LIN {X 0,Y 516.884,Z 407.102,A -85,B 0,C 180,E1 -5001.284,E2 -5001.284} C_VEL
LIN {X 0,Y 516.874,Z 407.103,A -85,B 0,C 180,E1 -5004.22,E2 -5004.22} C_VEL
LIN {X 0,Y 516.899,Z 407.102,A -85,B 0,C 180,E1 -5007.053,E2 -5007.053} C_VEL
LIN {X 0,Y 516.896,Z 407.098,A -85,B 0,C 180,E1 -5009.796,E2 -5009.796} C_VEL
LIN {X 0,Y 516.931,Z 407.097,A -85,B 0,C 180,E1 -5012.467,E2 -5012.467} C_VEL
LIN {X 0,Y 516.878,Z 407.102,A -85,B 0,C 180,E1 -5015.07,E2 -5015.07} C_VEL
LIN {X 0,Y 516.871,Z 407.103,A -85,B 0,C 180,E1 -5017.621,E2 -5017.621} C_VEL
LIN {X 0,Y 516.936,Z 407.096,A -85,B 0,C 180,E1 -5020.13,E2 -5020.13} C_VEL
LIN {X 0,Y 516.935,Z 407.096,A -85,B 0,C 180,E1 -5022.596,E2 -5022.596} C_VEL
LIN {X 0,Y 516.946,Z 407.095,A -85,B 0,C 180,E1 -5025.03,E2 -5025.03} C_VEL
LIN {X 0,Y 517.008,Z 407.087,A -85,B 0,C 180,E1 -5028.235,E2 -5028.235} C_VEL
LIN {X 0,Y 516.961,Z 407.092,A -85,B 0,C 180,E1 -5031.399,E2 -5031.399} C_VEL
LIN {X 0,Y 517.013,Z 407.086,A -85,B 0,C 180,E1 -5033.757,E2 -5033.757} C_VEL
LIN {X 0,Y 517.087,Z 407.075,A -85,B 0,C 180,E1 -5037.663,E2 -5037.663} C_VEL
LIN {X 0,Y 517.098,Z 407.076,A -85,B 0,C 180,E1 -5040.779,E2 -5040.779} C_VEL
LIN {X 0,Y 517.019,Z 407.085,A -85,B 0,C 180,E1 -5043.117,E2 -5043.117} C_VEL
LIN {X 0,Y 517.014,Z 407.087,A -85,B 0,C 180,E1 -5046.243,E2 -5046.243} C_VEL
LIN {X 0,Y 516.945,Z 407.094,A -85,B 0,C 180,E1 -5049.389,E2 -5049.389} C_VEL
LIN {X 0,Y 516.987,Z 407.09,A -85,B 0,C 180,E1 -5051.824,E2 -5051.824} C_VEL
LIN {X 0,Y 516.948,Z 407.092,A -85,B 0,C 180,E1 -5055.147,E2 -5055.147} C_VEL
LIN {X 0,Y 516.93,Z 407.097,A -85,B 0,C 180,E1 -5058.222,E2 -5058.222} C_VEL
LIN {X 0,Y 516.916,Z 407.097,A -85,B 0,C 180,E1 -5060.701,E2 -5060.701} C_VEL
LIN {X 0,Y 516.893,Z 407.101,A -85,B 0,C 180,E1 -5064.073,E2 -5064.073} C_VEL
LIN {X 0,Y 516.929,Z 407.095,A -85,B 0,C 180,E1 -5066.658,E2 -5066.658} C_VEL
LIN {X 0,Y 516.914,Z 407.098,A -85,B 0,C 180,E1 -5069.524,E2 -5069.524} C_VEL
LIN {X 0,Y 516.904,Z 407.1,A -85,B 0,C 180,E1 -5072.544,E2 -5072.544} C_VEL
LIN {X 0,Y 516.884,Z 407.101,A -85,B 0,C 180,E1 -5075.332,E2 -5075.332} C_VEL
LIN {X 0,Y 516.884,Z 407.103,A -85,B 0,C 180,E1 -5077.943,E2 -5077.943} C_VEL
LIN {X 0,Y 516.885,Z 407.1,A -85,B 0,C 180,E1 -5080.742,E2 -5080.742} C_VEL
LIN {X 0,Y 516.907,Z 407.1,A -85,B 0,C 180,E1 -5082.829,E2 -5082.829} C_VEL
LIN {X 0,Y 516.925,Z 407.098,A -85,B 0,C 180,E1 -5085.01,E2 -5085.01} C_VEL
LIN {X 0,Y 516.926,Z 407.098,A -85,B 0,C 180,E1 -5088.398,E2 -5088.398} C_VEL
LIN {X 0,Y 516.897,Z 407.1,A -85,B 0,C 180,E1 -5091.588,E2 -5091.588} C_VEL
LIN {X 0,Y 518.558,Z 416.082,A -85,B 0,C 180,E1 -5093.875,E2 -5093.875} C_VEL
LIN {X 0,Y 518.241,Z 427.468,A -85,B 0,C 180,E1 -5096.453,E2 -5096.453} C_VEL
LIN {X 0,Y 518.028,Z 441.136,A -85,B 0,C 180,E1 -5099.419,E2 -5099.419} C_VEL
LIN {X 0,Y 517.802,Z 455.931,A -85,B 0,C 180,E1 -5102.518,E2 -5102.518} C_VEL
LIN {X 0,Y 517.585,Z 470.324,A -85,B 0,C 180,E1 -5105.472,E2 -5105.472} C_VEL
LIN {X 0,Y 517.369,Z 484.144,A -85,B 0,C 180,E1 -5108.274,E2 -5108.274} C_VEL
LIN {X 0,Y 517.16,Z 499.664,A -85,B 0,C 180,E1 -5111.376,E2 -5111.376} C_VEL
LIN {X 0,Y 516.923,Z 514.192,A -85,B 0,C 180,E1 -5114.222,E2 -5114.222} C_VEL
LIN {X 0,Y 516.797,Z 523.545,A -85,B 0,C 180,E1 -5116.057,E2 -5116.057} C_VEL
LIN {X 0,Y 518.494,Z 536.775,A -85,B 0,C 180,E1 -5116.378,E2 -5116.378} C_VEL
LIN {X 0,Y 518.195,Z 548.997,A -85,B 0,C 180,E1 -5116.77,E2 -5116.77} C_VEL
LIN {X 0,Y 517.989,Z 560.148,A -85,B 0,C 180,E1 -5117.263,E2 -5117.263} C_VEL
LIN {X 0,Y 517.733,Z 571.933,A -85,B 0,C 180,E1 -5117.938,E2 -5117.938} C_VEL
LIN {X 0,Y 517.41,Z 582.942,A -85,B 0,C 180,E1 -5118.74,E2 -5118.74} C_VEL
LIN {X 0,Y 517.136,Z 592.815,A -85,B 0,C 180,E1 -5119.626,E2 -5119.626} C_VEL
LIN {X 0,Y 516.877,Z 601.829,A -85,B 0,C 180,E1 -5120.609,E2 -5120.609} C_VEL
LIN {X 0,Y 516.655,Z 610.643,A -85,B 0,C 180,E1 -5121.788,E2 -5121.788} C_VEL
LIN {X 0,Y 516.507,Z 617.697,A -85,B 0,C 180,E1 -5122.966,E2 -5122.966} C_VEL
LIN {X 0,Y 516.454,Z 623.311,A -85,B 0,C 180,E1 -5124.142,E2 -5124.142} C_VEL
LIN {X 0,Y 516.271,Z 627.663,A -85,B 0,C 180,E1 -5125.315,E2 -5125.315} C_VEL
LIN {X 0,Y 516.354,Z 629.957,A -85,B 0,C 180,E1 -5126.098,E2 -5126.098} C_VEL
LIN {X 0,Y 516.282,Z 631.806,A -85,B 0,C 180,E1 -5126.879,E2 -5126.879} C_VEL
LIN {X 0,Y 516.261,Z 633.192,A -85,B 0,C 180,E1 -5127.659,E2 -5127.659} C_VEL
LIN {X 0,Y 516.16,Z 634.785,A -85,B 0,C 180,E1 -5129.22,E2 -5129.22} C_VEL
LIN {X 0,Y 516.154,Z 635,A -85,B 0,C 180,E1 -5130,E2 -5130} C_VEL
LIN {X 0,Y 516.192,Z 634.183,A -85,B 0,C 180,E1 -5131.56,E2 -5131.56} C_VEL
LIN {X 0,Y 516.261,Z 633.195,A -85,B 0,C 180,E1 -5132.341,E2 -5132.341} C_VEL
LIN {X 0,Y 516.282,Z 631.81,A -85,B 0,C 180,E1 -5133.121,E2 -5133.121} C_VEL
LIN {X 0,Y 516.344,Z 628.891,A -85,B 0,C 180,E1 -5134.293,E2 -5134.293} C_VEL
LIN {X 0,Y 516.405,Z 624.912,A -85,B 0,C 180,E1 -5135.467,E2 -5135.467} C_VEL
LIN {X 0,Y 516.479,Z 618.942,A -85,B 0,C 180,E1 -5136.797,E2 -5136.797} C_VEL
LIN {X 0,Y 516.617,Z 611.904,A -85,B 0,C 180,E1 -5138.016,E2 -5138.016} C_VEL
LIN {X 0,Y 516.825,Z 603.448,A -85,B 0,C 180,E1 -5139.194,E2 -5139.194} C_VEL
LIN {X 0,Y 517.058,Z 594.795,A -85,B 0,C 180,E1 -5140.178,E2 -5140.178} C_VEL
LIN {X 0,Y 517.393,Z 584.136,A -85,B 0,C 180,E1 -5141.161,E2 -5141.161} C_VEL
LIN {X 0,Y 517.651,Z 572.582,A -85,B 0,C 180,E1 -5142.019,E2 -5142.019} C_VEL
LIN {X 0,Y 517.968,Z 562.096,A -85,B 0,C 180,E1 -5142.638,E2 -5142.638} C_VEL
LIN {X 0,Y 518.188,Z 550.297,A -85,B 0,C 180,E1 -5143.181,E2 -5143.181} C_VEL
LIN {X 0,Y 518.464,Z 536.759,A -85,B 0,C 180,E1 -5143.623,E2 -5143.623} C_VEL
LIN {X 0,Y 516.797,Z 523.543,A -85,B 0,C 180,E1 -5143.943,E2 -5143.943} C_VEL
LIN {X 0,Y 517.079,Z 506.87,A -85,B 0,C 180,E1 -5147.195,E2 -5147.195} C_VEL
LIN {X 0,Y 517.213,Z 492.186,A -85,B 0,C 180,E1 -5150.11,E2 -5150.11} C_VEL
LIN {X 0,Y 517.513,Z 476.876,A -85,B 0,C 180,E1 -5153.193,E2 -5153.193} C_VEL
LIN {X 0,Y 517.711,Z 461.343,A -85,B 0,C 180,E1 -5156.368,E2 -5156.368} C_VEL
LIN {X 0,Y 517.924,Z 447.472,A -85,B 0,C 180,E1 -5159.243,E2 -5159.243} C_VEL
LIN {X 0,Y 518.112,Z 434.804,A -85,B 0,C 180,E1 -5161.94,E2 -5161.94} C_VEL
LIN {X 0,Y 518.506,Z 420.311,A -85,B 0,C 180,E1 -5165.148,E2 -5165.148} C_VEL
LIN {X 0,Y 518.426,Z 415.032,A -85,B 0,C 180,E1 -5166.377,E2 -5166.377} C_VEL
LIN {X 0,Y 516.898,Z 407.101,A -85,B 0,C 180,E1 -5168.412,E2 -5168.412} C_VEL
LIN {X 0,Y 516.926,Z 407.095,A -85,B 0,C 180,E1 -5171.603,E2 -5171.603} C_VEL
LIN {X 0,Y 516.926,Z 407.096,A -85,B 0,C 180,E1 -5175.01,E2 -5175.01} C_VEL
LIN {X 0,Y 516.919,Z 407.098,A -85,B 0,C 180,E1 -5178.398,E2 -5178.398} C_VEL
LIN {X 0,Y 516.884,Z 407.101,A -85,B 0,C 180,E1 -5181.284,E2 -5181.284} C_VEL
LIN {X 0,Y 516.893,Z 407.101,A -85,B 0,C 180,E1 -5184.221,E2 -5184.221} C_VEL
LIN {X 0,Y 516.902,Z 407.099,A -85,B 0,C 180,E1 -5187.053,E2 -5187.053} C_VEL
LIN {X 0,Y 516.897,Z 407.1,A -85,B 0,C 180,E1 -5189.796,E2 -5189.796} C_VEL
LIN {X 0,Y 516.932,Z 407.096,A -85,B 0,C 180,E1 -5192.467,E2 -5192.467} C_VEL
LIN {X 0,Y 516.879,Z 407.101,A -85,B 0,C 180,E1 -5195.07,E2 -5195.07} C_VEL
LIN {X 0,Y 516.872,Z 407.103,A -85,B 0,C 180,E1 -5197.622,E2 -5197.622} C_VEL
LIN {X 0,Y 516.937,Z 407.095,A -85,B 0,C 180,E1 -5200.13,E2 -5200.13} C_VEL
LIN {X 0,Y 516.936,Z 407.094,A -85,B 0,C 180,E1 -5202.596,E2 -5202.596} C_VEL
LIN {X 0,Y 516.947,Z 407.093,A -85,B 0,C 180,E1 -5205.03,E2 -5205.03} C_VEL
LIN {X 0,Y 517.009,Z 407.087,A -85,B 0,C 180,E1 -5208.235,E2 -5208.235} C_VEL
LIN {X 0,Y 516.96,Z 407.092,A -85,B 0,C 180,E1 -5211.4,E2 -5211.4} C_VEL
LIN {X 0,Y 517.015,Z 407.087,A -85,B 0,C 180,E1 -5213.757,E2 -5213.757} C_VEL
LIN {X 0,Y 517.09,Z 407.077,A -85,B 0,C 180,E1 -5217.663,E2 -5217.663} C_VEL
LIN {X 0,Y 517.1,Z 407.073,A -85,B 0,C 180,E1 -5220.779,E2 -5220.779} C_VEL
LIN {X 0,Y 517.018,Z 407.085,A -85,B 0,C 180,E1 -5223.117,E2 -5223.117} C_VEL
LIN {X 0,Y 517.014,Z 407.086,A -85,B 0,C 180,E1 -5226.243,E2 -5226.243} C_VEL
LIN {X 0,Y 516.953,Z 407.094,A -85,B 0,C 180,E1 -5229.389,E2 -5229.389} C_VEL
LIN {X 0,Y 516.989,Z 407.089,A -85,B 0,C 180,E1 -5231.824,E2 -5231.824} C_VEL
LIN {X 0,Y 516.949,Z 407.095,A -85,B 0,C 180,E1 -5235.147,E2 -5235.147} C_VEL
LIN {X 0,Y 516.93,Z 407.095,A -85,B 0,C 180,E1 -5238.222,E2 -5238.222} C_VEL
LIN {X 0,Y 516.917,Z 407.097,A -85,B 0,C 180,E1 -5240.701,E2 -5240.701} C_VEL
LIN {X 0,Y 516.907,Z 407.098,A -85,B 0,C 180,E1 -5244.072,E2 -5244.072} C_VEL
LIN {X 0,Y 516.93,Z 407.096,A -85,B 0,C 180,E1 -5246.658,E2 -5246.658} C_VEL
LIN {X 0,Y 516.916,Z 407.099,A -85,B 0,C 180,E1 -5249.524,E2 -5249.524} C_VEL
LIN {X 0,Y 516.905,Z 407.098,A -85,B 0,C 180,E1 -5252.544,E2 -5252.544} C_VEL
LIN {X 0,Y 516.87,Z 407.104,A -85,B 0,C 180,E1 -5255.33,E2 -5255.33} C_VEL
LIN {X 0,Y 516.883,Z 407.102,A -85,B 0,C 180,E1 -5257.943,E2 -5257.943} C_VEL
LIN {X 0,Y 516.888,Z 407.101,A -85,B 0,C 180,E1 -5260.741,E2 -5260.741} C_VEL
LIN {X 0,Y 516.909,Z 407.099,A -85,B 0,C 180,E1 -5262.829,E2 -5262.829} C_VEL
LIN {X 0,Y 516.927,Z 407.097,A -85,B 0,C 180,E1 -5265.01,E2 -5265.01} C_VEL
LIN {X 0,Y 516.927,Z 407.095,A -85,B 0,C 180,E1 -5268.397,E2 -5268.397} C_VEL
LIN {X 0,Y 516.915,Z 407.097,A -85,B 0,C 180,E1 -5270.299,E2 -5270.299} C_VEL
LIN {X 0,Y 516.245,Z 407.183,A -85,B 0,C 180,E1 -5270.949,E2 -5270.949} C_VEL
LIN {X 0,Y 513.386,Z 407.538,A -85,B 0,C 180,E1 -5272.004,E2 -5272.004} C_VEL
LIN {X 0,Y 510.964,Z 407.84,A -85,B 0,C 180,E1 -5272.854,E2 -5272.854} C_VEL
LIN {X 0,Y 509.914,Z 407.969,A -85,B 0,C 180,E1 -5273.51,E2 -5273.51} C_VEL
LIN {X 0,Y 509.824,Z 407.98,A -85,B 0,C 180,E1 -5273.733,E2 -5273.733} C_VEL
LIN {X 0,Y 509.863,Z 407.977,A -85,B 0,C 180,E1 -5276.539,E2 -5276.539} C_VEL
LIN {X 0,Y 509.849,Z 407.979,A -85,B 0,C 180,E1 -5279.334,E2 -5279.334} C_VEL
LIN {X 0,Y 509.898,Z 407.97,A -85,B 0,C 180,E1 -5282.055,E2 -5282.055} C_VEL
LIN {X 0,Y 509.882,Z 407.976,A -85,B 0,C 180,E1 -5284.704,E2 -5284.704} C_VEL
LIN {X 0,Y 509.841,Z 407.978,A -85,B 0,C 180,E1 -5287.455,E2 -5287.455} C_VEL
LIN {X 0,Y 509.921,Z 407.968,A -85,B 0,C 180,E1 -5289.845,E2 -5289.845} C_VEL
LIN {X 0,Y 509.886,Z 407.975,A -85,B 0,C 180,E1 -5293.175,E2 -5293.175} C_VEL
LIN {X 0,Y 509.868,Z 407.976,A -85,B 0,C 180,E1 -5295.634,E2 -5295.634} C_VEL
LIN {X 0,Y 509.88,Z 407.975,A -85,B 0,C 180,E1 -5296.677,E2 -5296.677} C_VEL
LIN {X 0,Y 511.479,Z 413.745,A -85,B 0,C 180,E1 -5296.997,E2 -5296.997} C_VEL
LIN {X 0,Y 511.344,Z 424.626,A -85,B 0,C 180,E1 -5297.607,E2 -5297.607} C_VEL
LIN {X 0,Y 511.051,Z 435.759,A -85,B 0,C 180,E1 -5298.397,E2 -5298.397} C_VEL
LIN {X 0,Y 510.75,Z 445.883,A -85,B 0,C 180,E1 -5299.294,E2 -5299.294} C_VEL
LIN {X 0,Y 510.417,Z 454.958,A -85,B 0,C 180,E1 -5300.289,E2 -5300.289} C_VEL
LIN {X 0,Y 510.088,Z 463.74,A -85,B 0,C 180,E1 -5301.482,E2 -5301.482} C_VEL
LIN {X 0,Y 509.898,Z 470.788,A -85,B 0,C 180,E1 -5302.675,E2 -5302.675} C_VEL
LIN {X 0,Y 509.762,Z 475.541,A -85,B 0,C 180,E1 -5303.668,E2 -5303.668} C_VEL
LIN {X 0,Y 509.556,Z 480.164,A -85,B 0,C 180,E1 -5304.856,E2 -5304.856} C_VEL
LIN {X 0,Y 509.517,Z 483.685,A -85,B 0,C 180,E1 -5306.045,E2 -5306.045} C_VEL
LIN {X 0,Y 509.452,Z 485.511,A -85,B 0,C 180,E1 -5306.837,E2 -5306.837} C_VEL
LIN {X 0,Y 509.368,Z 486.894,A -85,B 0,C 180,E1 -5307.628,E2 -5307.628} C_VEL
LIN {X 0,Y 509.32,Z 488.474,A -85,B 0,C 180,E1 -5309.209,E2 -5309.209} C_VEL
LIN {X 0,Y 509.31,Z 488.707,A -85,B 0,C 180,E1 -5310,E2 -5310} C_VEL
LIN {X 0,Y 509.359,Z 487.954,A -85,B 0,C 180,E1 -5311.581,E2 -5311.581} C_VEL
LIN {X 0,Y 509.448,Z 485.687,A -85,B 0,C 180,E1 -5313.163,E2 -5313.163} C_VEL
LIN {X 0,Y 509.561,Z 482.884,A -85,B 0,C 180,E1 -5314.35,E2 -5314.35} C_VEL
LIN {X 0,Y 509.634,Z 479.091,A -85,B 0,C 180,E1 -5315.539,E2 -5315.539} C_VEL
LIN {X 0,Y 509.756,Z 473.172,A -85,B 0,C 180,E1 -5316.943,E2 -5316.943} C_VEL
LIN {X 0,Y 510.053,Z 465.599,A -85,B 0,C 180,E1 -5318.319,E2 -5318.319} C_VEL
LIN {X 0,Y 510.352,Z 457.266,A -85,B 0,C 180,E1 -5319.512,E2 -5319.512} C_VEL
LIN {X 0,Y 510.62,Z 448.688,A -85,B 0,C 180,E1 -5320.508,E2 -5320.508} C_VEL
LIN {X 0,Y 510.971,Z 438.097,A -85,B 0,C 180,E1 -5321.504,E2 -5321.504} C_VEL
LIN {X 0,Y 511.234,Z 428.336,A -85,B 0,C 180,E1 -5322.243,E2 -5322.243} C_VEL
LIN {X 0,Y 511.525,Z 417.45,A -85,B 0,C 180,E1 -5322.901,E2 -5322.901} C_VEL
LIN {X 0,Y 511.437,Z 413.548,A -85,B 0,C 180,E1 -5323.105,E2 -5323.105} C_VEL
LIN {X 0,Y 509.885,Z 407.973,A -85,B 0,C 180,E1 -5323.425,E2 -5323.425} C_VEL
LIN {X 0,Y 509.856,Z 407.977,A -85,B 0,C 180,E1 -5326.003,E2 -5326.003} C_VEL
LIN {X 0,Y 509.865,Z 407.974,A -85,B 0,C 180,E1 -5328.484,E2 -5328.484} C_VEL
LIN {X 0,Y 509.854,Z 407.978,A -85,B 0,C 180,E1 -5331.002,E2 -5331.002} C_VEL
LIN {X 0,Y 509.841,Z 407.979,A -85,B 0,C 180,E1 -5333.563,E2 -5333.563} C_VEL
LIN {X 0,Y 509.918,Z 407.969,A -85,B 0,C 180,E1 -5336.379,E2 -5336.379} C_VEL
LIN {X 0,Y 509.881,Z 407.975,A -85,B 0,C 180,E1 -5338.844,E2 -5338.844} C_VEL
LIN {X 0,Y 509.823,Z 407.983,A -85,B 0,C 180,E1 -5341.59,E2 -5341.59} C_VEL
LIN {X 0,Y 509.857,Z 407.976,A -85,B 0,C 180,E1 -5344.413,E2 -5344.413} C_VEL
LIN {X 0,Y 509.823,Z 407.981,A -85,B 0,C 180,E1 -5347.34,E2 -5347.34} C_VEL
LIN {X 0,Y 509.865,Z 407.976,A -85,B 0,C 180,E1 -5350.38,E2 -5350.38} C_VEL
LIN {X 0,Y 509.843,Z 407.979,A -85,B 0,C 180,E1 -5353.064,E2 -5353.064} C_VEL
LIN {X 0,Y 509.834,Z 407.978,A -85,B 0,C 180,E1 -5355.792,E2 -5355.792} C_VEL
LIN {X 0,Y 509.86,Z 407.977,A -85,B 0,C 180,E1 -5358.575,E2 -5358.575} C_VEL
LIN {X 0,Y 509.854,Z 407.977,A -85,B 0,C 180,E1 -5361.786,E2 -5361.786} C_VEL
LIN {X 0,Y 509.833,Z 407.98,A -85,B 0,C 180,E1 -5364.622,E2 -5364.622} C_VEL
LIN {X 0,Y 509.866,Z 407.975,A -85,B 0,C 180,E1 -5367.481,E2 -5367.481} C_VEL
LIN {X 0,Y 509.861,Z 407.976,A -85,B 0,C 180,E1 -5370.274,E2 -5370.274} C_VEL
LIN {X 0,Y 509.888,Z 407.973,A -85,B 0,C 180,E1 -5372.944,E2 -5372.944} C_VEL
LIN {X 0,Y 509.854,Z 407.977,A -85,B 0,C 180,E1 -5375.573,E2 -5375.573} C_VEL
LIN {X 0,Y 509.825,Z 407.981,A -85,B 0,C 180,E1 -5378.149,E2 -5378.149} C_VEL
LIN {X 0,Y 509.869,Z 407.976,A -85,B 0,C 180,E1 -5380.682,E2 -5380.682} C_VEL
LIN {X 0,Y 509.89,Z 407.972,A -85,B 0,C 180,E1 -5383.175,E2 -5383.175} C_VEL
LIN {X 0,Y 509.868,Z 407.974,A -85,B 0,C 180,E1 -5385.634,E2 -5385.634} C_VEL
LIN {X 0,Y 509.926,Z 407.968,A -85,B 0,C 180,E1 -5388.875,E2 -5388.875} C_VEL
LIN {X 0,Y 509.925,Z 407.968,A -85,B 0,C 180,E1 -5392.078,E2 -5392.078} C_VEL
LIN {X 0,Y 509.985,Z 407.962,A -85,B 0,C 180,E1 -5394.464,E2 -5394.464} C_VEL
LIN {X 0,Y 510.058,Z 407.951,A -85,B 0,C 180,E1 -5397.631,E2 -5397.631} C_VEL
LIN {X 0,Y 510.068,Z 407.952,A -85,B 0,C 180,E1 -5400.789,E2 -5400.789} C_VEL
LIN {X 0,Y 509.961,Z 407.964,A -85,B 0,C 180,E1 -5403.16,E2 -5403.16} C_VEL
LIN {X 0,Y 509.982,Z 407.963,A -85,B 0,C 180,E1 -5406.33,E2 -5406.33} C_VEL
LIN {X 0,Y 509.886,Z 407.973,A -85,B 0,C 180,E1 -5409.521,E2 -5409.521} C_VEL
LIN {X 0,Y 509.955,Z 407.965,A -85,B 0,C 180,E1 -5411.93,E2 -5411.93} C_VEL
LIN {X 0,Y 509.897,Z 407.97,A -85,B 0,C 180,E1 -5415.242,E2 -5415.242} C_VEL
LIN {X 0,Y 509.892,Z 407.974,A -85,B 0,C 180,E1 -5418.001,E2 -5418.001} C_VEL
LIN {X 0,Y 509.854,Z 407.977,A -85,B 0,C 180,E1 -5421.002,E2 -5421.002} C_VEL
LIN {X 0,Y 509.825,Z 407.981,A -85,B 0,C 180,E1 -5423.564,E2 -5423.564} C_VEL
LIN {X 0,Y 509.915,Z 407.971,A -85,B 0,C 180,E1 -5426.379,E2 -5426.379} C_VEL
LIN {X 0,Y 509.88,Z 407.972,A -85,B 0,C 180,E1 -5428.844,E2 -5428.844} C_VEL
LIN {X 0,Y 509.829,Z 407.98,A -85,B 0,C 180,E1 -5431.59,E2 -5431.59} C_VEL
LIN {X 0,Y 509.855,Z 407.977,A -85,B 0,C 180,E1 -5434.413,E2 -5434.413} C_VEL
LIN {X 0,Y 509.822,Z 407.982,A -85,B 0,C 180,E1 -5437.341,E2 -5437.341} C_VEL
LIN {X 0,Y 509.84,Z 407.979,A -85,B 0,C 180,E1 -5440.382,E2 -5440.382} C_VEL
LIN {X 0,Y 509.842,Z 407.981,A -85,B 0,C 180,E1 -5443.064,E2 -5443.064} C_VEL
LIN {X 0,Y 509.833,Z 407.98,A -85,B 0,C 180,E1 -5445.792,E2 -5445.792} C_VEL
LIN {X 0,Y 509.869,Z 407.977,A -85,B 0,C 180,E1 -5448.576,E2 -5448.576} C_VEL
LIN {X 0,Y 509.891,Z 408.122,A -85,B 0,C 180,E1 -5451.413,E2 -5451.413} C_VEL
LIN {X 0,Y 511.639,Z 417.468,A -85,B 0,C 180,E1 -5453.796,E2 -5453.796} C_VEL
LIN {X 0,Y 511.317,Z 427.794,A -85,B 0,C 180,E1 -5456.174,E2 -5456.174} C_VEL
LIN {X 0,Y 511.063,Z 441.426,A -85,B 0,C 180,E1 -5459.186,E2 -5459.186} C_VEL
LIN {X 0,Y 510.808,Z 456.196,A -85,B 0,C 180,E1 -5462.332,E2 -5462.332} C_VEL
LIN {X 0,Y 510.541,Z 470.48,A -85,B 0,C 180,E1 -5465.305,E2 -5465.305} C_VEL
LIN {X 0,Y 510.337,Z 483.348,A -85,B 0,C 180,E1 -5467.959,E2 -5467.959} C_VEL
LIN {X 0,Y 510.095,Z 497.76,A -85,B 0,C 180,E1 -5470.9,E2 -5470.9} C_VEL
LIN {X 0,Y 509.894,Z 511.103,A -85,B 0,C 180,E1 -5473.587,E2 -5473.587} C_VEL
LIN {X 0,Y 509.777,Z 522.516,A -85,B 0,C 180,E1 -5475.861,E2 -5475.861} C_VEL
LIN {X 0,Y 510.845,Z 532.053,A -85,B 0,C 180,E1 -5476.078,E2 -5476.078} C_VEL
LIN {X 0,Y 511.513,Z 538.516,A -85,B 0,C 180,E1 -5476.265,E2 -5476.265} C_VEL
LIN {X 0,Y 511.199,Z 551.66,A -85,B 0,C 180,E1 -5476.737,E2 -5476.737} C_VEL
LIN {X 0,Y 510.865,Z 564.127,A -85,B 0,C 180,E1 -5477.356,E2 -5477.356} C_VEL
LIN {X 0,Y 510.599,Z 575.475,A -85,B 0,C 180,E1 -5478.085,E2 -5478.085} C_VEL
LIN {X 0,Y 510.221,Z 586.551,A -85,B 0,C 180,E1 -5478.982,E2 -5478.982} C_VEL
LIN {X 0,Y 509.947,Z 595.605,A -85,B 0,C 180,E1 -5479.88,E2 -5479.88} C_VEL
LIN {X 0,Y 509.708,Z 605.469,A -85,B 0,C 180,E1 -5481.076,E2 -5481.076} C_VEL
LIN {X 0,Y 509.513,Z 613.341,A -85,B 0,C 180,E1 -5482.271,E2 -5482.271} C_VEL
LIN {X 0,Y 509.344,Z 620.603,A -85,B 0,C 180,E1 -5483.663,E2 -5483.663} C_VEL
LIN {X 0,Y 509.276,Z 625.448,A -85,B 0,C 180,E1 -5484.854,E2 -5484.854} C_VEL
LIN {X 0,Y 509.286,Z 629.162,A -85,B 0,C 180,E1 -5486.044,E2 -5486.044} C_VEL
LIN {X 0,Y 509.231,Z 631.07,A -85,B 0,C 180,E1 -5486.835,E2 -5486.835} C_VEL
LIN {X 0,Y 509.189,Z 632.501,A -85,B 0,C 180,E1 -5487.627,E2 -5487.627} C_VEL
LIN {X 0,Y 509.089,Z 634.138,A -85,B 0,C 180,E1 -5489.209,E2 -5489.209} C_VEL
LIN {X 0,Y 509.083,Z 634.36,A -85,B 0,C 180,E1 -5490,E2 -5490} C_VEL
LIN {X 0,Y 509.089,Z 634.138,A -85,B 0,C 180,E1 -5490.791,E2 -5490.791} C_VEL
LIN {X 0,Y 509.189,Z 632.504,A -85,B 0,C 180,E1 -5492.373,E2 -5492.373} C_VEL
LIN {X 0,Y 509.231,Z 631.073,A -85,B 0,C 180,E1 -5493.165,E2 -5493.165} C_VEL
LIN {X 0,Y 509.269,Z 628.06,A -85,B 0,C 180,E1 -5494.353,E2 -5494.353} C_VEL
LIN {X 0,Y 509.344,Z 623.985,A -85,B 0,C 180,E1 -5495.543,E2 -5495.543} C_VEL
LIN {X 0,Y 509.403,Z 618.179,A -85,B 0,C 180,E1 -5496.845,E2 -5496.845} C_VEL
LIN {X 0,Y 509.563,Z 610.885,A -85,B 0,C 180,E1 -5498.127,E2 -5498.127} C_VEL
LIN {X 0,Y 509.774,Z 602.427,A -85,B 0,C 180,E1 -5499.323,E2 -5499.323} C_VEL
LIN {X 0,Y 510.031,Z 593.774,A -85,B 0,C 180,E1 -5500.319,E2 -5500.319} C_VEL
LIN {X 0,Y 510.379,Z 583.113,A -85,B 0,C 180,E1 -5501.316,E2 -5501.316} C_VEL
LIN {X 0,Y 510.619,Z 571.554,A -85,B 0,C 180,E1 -5502.187,E2 -5502.187} C_VEL
LIN {X 0,Y 510.963,Z 561.069,A -85,B 0,C 180,E1 -5502.814,E2 -5502.814} C_VEL
LIN {X 0,Y 511.229,Z 549.274,A -85,B 0,C 180,E1 -5503.364,E2 -5503.364} C_VEL
LIN {X 0,Y 511.464,Z 536.19,A -85,B 0,C 180,E1 -5503.8,E2 -5503.8} C_VEL
LIN {X 0,Y 509.873,Z 524.402,A -85,B 0,C 180,E1 -5504.098,E2 -5504.098} C_VEL
LIN {X 0,Y 509.766,Z 522.385,A -85,B 0,C 180,E1 -5504.165,E2 -5504.165} C_VEL
LIN {X 0,Y 509.999,Z 505.962,A -85,B 0,C 180,E1 -5507.441,E2 -5507.441} C_VEL
LIN {X 0,Y 510.207,Z 490.878,A -85,B 0,C 180,E1 -5510.497,E2 -5510.497} C_VEL
LIN {X 0,Y 510.462,Z 476.097,A -85,B 0,C 180,E1 -5513.533,E2 -5513.533} C_VEL
LIN {X 0,Y 510.708,Z 461.509,A -85,B 0,C 180,E1 -5516.557,E2 -5516.557} C_VEL
LIN {X 0,Y 510.945,Z 447.746,A -85,B 0,C 180,E1 -5519.455,E2 -5519.455} C_VEL
LIN {X 0,Y 511.175,Z 434.056,A -85,B 0,C 180,E1 -5522.426,E2 -5522.426} C_VEL
LIN {X 0,Y 511.637,Z 420.237,A -85,B 0,C 180,E1 -5525.551,E2 -5525.551} C_VEL
LIN {X 0,Y 511.643,Z 417.453,A -85,B 0,C 180,E1 -5526.204,E2 -5526.204} C_VEL
LIN {X 0,Y 509.889,Z 407.973,A -85,B 0,C 180,E1 -5528.65,E2 -5528.65} C_VEL
LIN {X 0,Y 509.865,Z 407.974,A -85,B 0,C 180,E1 -5531.897,E2 -5531.897} C_VEL
LIN {X 0,Y 509.86,Z 407.977,A -85,B 0,C 180,E1 -5535.332,E2 -5535.332} C_VEL
LIN {X 0,Y 509.861,Z 407.978,A -85,B 0,C 180,E1 -5538.575,E2 -5538.575} C_VEL
LIN {X 0,Y 509.855,Z 407.978,A -85,B 0,C 180,E1 -5541.786,E2 -5541.786} C_VEL
LIN {X 0,Y 509.848,Z 407.978,A -85,B 0,C 180,E1 -5544.623,E2 -5544.623} C_VEL
LIN {X 0,Y 509.87,Z 407.976,A -85,B 0,C 180,E1 -5547.481,E2 -5547.481} C_VEL
LIN {X 0,Y 509.862,Z 407.978,A -85,B 0,C 180,E1 -5550.274,E2 -5550.274} C_VEL
LIN {X 0,Y 509.889,Z 407.971,A -85,B 0,C 180,E1 -5552.945,E2 -5552.945} C_VEL
LIN {X 0,Y 509.855,Z 407.978,A -85,B 0,C 180,E1 -5555.573,E2 -5555.573} C_VEL
LIN {X 0,Y 509.826,Z 407.981,A -85,B 0,C 180,E1 -5558.149,E2 -5558.149} C_VEL
LIN {X 0,Y 509.87,Z 407.975,A -85,B 0,C 180,E1 -5560.682,E2 -5560.682} C_VEL
LIN {X 0,Y 509.891,Z 407.973,A -85,B 0,C 180,E1 -5563.175,E2 -5563.175} C_VEL
LIN {X 0,Y 509.869,Z 407.976,A -85,B 0,C 180,E1 -5565.634,E2 -5565.634} C_VEL
LIN {X 0,Y 509.926,Z 407.967,A -85,B 0,C 180,E1 -5568.875,E2 -5568.875} C_VEL
LIN {X 0,Y 509.925,Z 407.968,A -85,B 0,C 180,E1 -5572.078,E2 -5572.078} C_VEL
LIN {X 0,Y 509.987,Z 407.961,A -85,B 0,C 180,E1 -5574.464,E2 -5574.464} C_VEL
LIN {X 0,Y 510.061,Z 407.952,A -85,B 0,C 180,E1 -5577.631,E2 -5577.631} C_VEL
LIN {X 0,Y 510.07,Z 407.948,A -85,B 0,C 180,E1 -5580.79,E2 -5580.79} C_VEL
LIN {X 0,Y 509.96,Z 407.964,A -85,B 0,C 180,E1 -5583.16,E2 -5583.16} C_VEL
LIN {X 0,Y 509.964,Z 407.964,A -85,B 0,C 180,E1 -5586.33,E2 -5586.33} C_VEL
LIN {X 0,Y 509.894,Z 407.974,A -85,B 0,C 180,E1 -5589.52,E2 -5589.52} C_VEL
LIN {X 0,Y 509.956,Z 407.964,A -85,B 0,C 180,E1 -5591.931,E2 -5591.931} C_VEL
LIN {X 0,Y 509.898,Z 407.972,A -85,B 0,C 180,E1 -5595.242,E2 -5595.242} C_VEL
LIN {X 0,Y 509.893,Z 407.973,A -85,B 0,C 180,E1 -5598.001,E2 -5598.001} C_VEL
LIN {X 0,Y 509.855,Z 407.977,A -85,B 0,C 180,E1 -5601.002,E2 -5601.002} C_VEL
LIN {X 0,Y 509.868,Z 407.975,A -85,B 0,C 180,E1 -5604.426,E2 -5604.426} C_VEL
LIN {X 0,Y 509.889,Z 407.973,A -85,B 0,C 180,E1 -5607.056,E2 -5607.056} C_VEL
LIN {X 0,Y 509.861,Z 407.977,A -85,B 0,C 180,E1 -5609.751,E2 -5609.751} C_VEL
LIN {X 0,Y 509.881,Z 407.974,A -85,B 0,C 180,E1 -5612.775,E2 -5612.775} C_VEL
LIN {X 0,Y 509.83,Z 407.98,A -85,B 0,C 180,E1 -5615.578,E2 -5615.578} C_VEL
LIN {X 0,Y 509.853,Z 407.977,A -85,B 0,C 180,E1 -5618.338,E2 -5618.338} C_VEL
LIN {X 0,Y 509.861,Z 407.977,A -85,B 0,C 180,E1 -5621.425,E2 -5621.425} C_VEL
LIN {X 0,Y 509.861,Z 407.978,A -85,B 0,C 180,E1 -5624.668,E2 -5624.668} C_VEL
LIN {X 0,Y 509.868,Z 407.975,A -85,B 0,C 180,E1 -5628.102,E2 -5628.102} C_VEL
LIN {X 0,Y 509.881,Z 407.974,A -85,B 0,C 180,E1 -5630.65,E2 -5630.65} C_VEL
LIN {X 0,Y 509.824,Z 407.98,A -85,B 0,C 180,E1 -5633.733,E2 -5633.733} C_VEL
LIN {X 0,Y 509.156,Z 408.065,A -85,B 0,C 180,E1 -5634.392,E2 -5634.392} C_VEL
LIN {X 0,Y 506.344,Z 408.416,A -85,B 0,C 180,E1 -5635.464,E2 -5635.464} C_VEL
LIN {X 0,Y 503.957,Z 408.714,A -85,B 0,C 180,E1 -5636.328,E2 -5636.328} C_VEL
LIN {X 0,Y 502.91,Z 408.843,A -85,B 0,C 180,E1 -5636.994,E2 -5636.994} C_VEL
LIN {X 0,Y 502.812,Z 408.853,A -85,B 0,C 180,E1 -5637.22,E2 -5637.22} C_VEL
LIN {X 0,Y 502.819,Z 408.852,A -85,B 0,C 180,E1 -5640.065,E2 -5640.065} C_VEL
LIN {X 0,Y 502.838,Z 408.852,A -85,B 0,C 180,E1 -5642.533,E2 -5642.533} C_VEL
LIN {X 0,Y 502.833,Z 408.852,A -85,B 0,C 180,E1 -5645.298,E2 -5645.298} C_VEL
LIN {X 0,Y 502.789,Z 408.857,A -85,B 0,C 180,E1 -5647.827,E2 -5647.827} C_VEL
LIN {X 0,Y 502.828,Z 408.853,A -85,B 0,C 180,E1 -5650.4,E2 -5650.4} C_VEL
LIN {X 0,Y 502.834,Z 408.853,A -85,B 0,C 180,E1 -5652.931,E2 -5652.931} C_VEL
LIN {X 0,Y 502.849,Z 408.851,A -85,B 0,C 180,E1 -5655.429,E2 -5655.429} C_VEL
LIN {X 0,Y 502.845,Z 409.01,A -85,B 0,C 180,E1 -5656.487,E2 -5656.487} C_VEL
LIN {X 0,Y 504.491,Z 414.784,A -85,B 0,C 180,E1 -5656.814,E2 -5656.814} C_VEL
LIN {X 0,Y 504.501,Z 424.331,A -85,B 0,C 180,E1 -5657.35,E2 -5657.35} C_VEL
LIN {X 0,Y 504.208,Z 435.502,A -85,B 0,C 180,E1 -5658.135,E2 -5658.135} C_VEL
LIN {X 0,Y 503.886,Z 445.846,A -85,B 0,C 180,E1 -5659.045,E2 -5659.045} C_VEL
LIN {X 0,Y 503.554,Z 454.289,A -85,B 0,C 180,E1 -5659.953,E2 -5659.953} C_VEL
LIN {X 0,Y 503.295,Z 462.043,A -85,B 0,C 180,E1 -5660.962,E2 -5660.962} C_VEL
LIN {X 0,Y 502.988,Z 469.625,A -85,B 0,C 180,E1 -5662.17,E2 -5662.17} C_VEL
LIN {X 0,Y 502.783,Z 476.548,A -85,B 0,C 180,E1 -5663.579,E2 -5663.579} C_VEL
LIN {X 0,Y 502.561,Z 481.171,A -85,B 0,C 180,E1 -5664.785,E2 -5664.785} C_VEL
LIN {X 0,Y 502.506,Z 484.692,A -85,B 0,C 180,E1 -5665.99,E2 -5665.99} C_VEL
LIN {X 0,Y 502.434,Z 486.518,A -85,B 0,C 180,E1 -5666.792,E2 -5666.792} C_VEL
LIN {X 0,Y 502.346,Z 487.9,A -85,B 0,C 180,E1 -5667.594,E2 -5667.594} C_VEL
LIN {X 0,Y 502.299,Z 489.478,A -85,B 0,C 180,E1 -5669.198,E2 -5669.198} C_VEL
LIN {X 0,Y 502.286,Z 489.711,A -85,B 0,C 180,E1 -5670,E2 -5670} C_VEL
LIN {X 0,Y 502.346,Z 488.957,A -85,B 0,C 180,E1 -5671.603,E2 -5671.603} C_VEL
LIN {X 0,Y 502.43,Z 486.691,A -85,B 0,C 180,E1 -5673.207,E2 -5673.207} C_VEL
LIN {X 0,Y 502.554,Z 483.887,A -85,B 0,C 180,E1 -5674.411,E2 -5674.411} C_VEL
LIN {X 0,Y 502.649,Z 480.093,A -85,B 0,C 180,E1 -5675.617,E2 -5675.617} C_VEL
LIN {X 0,Y 502.78,Z 474.179,A -85,B 0,C 180,E1 -5677.039,E2 -5677.039} C_VEL
LIN {X 0,Y 503.078,Z 467.798,A -85,B 0,C 180,E1 -5678.233,E2 -5678.233} C_VEL
LIN {X 0,Y 503.368,Z 459.788,A -85,B 0,C 180,E1 -5679.442,E2 -5679.442} C_VEL
LIN {X 0,Y 503.628,Z 451.577,A -85,B 0,C 180,E1 -5680.452,E2 -5680.452} C_VEL
LIN {X 0,Y 504.026,Z 441.4,A -85,B 0,C 180,E1 -5681.461,E2 -5681.461} C_VEL
LIN {X 0,Y 504.371,Z 430.927,A -85,B 0,C 180,E1 -5682.296,E2 -5682.296} C_VEL
LIN {X 0,Y 504.629,Z 420.251,A -85,B 0,C 180,E1 -5682.978,E2 -5682.978} C_VEL
LIN {X 0,Y 504.695,Z 416.483,A -85,B 0,C 180,E1 -5683.181,E2 -5683.181} C_VEL
LIN {X 0,Y 502.825,Z 408.85,A -85,B 0,C 180,E1 -5683.617,E2 -5683.617} C_VEL
LIN {X 0,Y 502.821,Z 408.853,A -85,B 0,C 180,E1 -5686.233,E2 -5686.233} C_VEL
LIN {X 0,Y 502.83,Z 408.851,A -85,B 0,C 180,E1 -5688.752,E2 -5688.752} C_VEL
LIN {X 0,Y 502.787,Z 408.859,A -85,B 0,C 180,E1 -5691.311,E2 -5691.311} C_VEL
LIN {X 0,Y 502.796,Z 408.856,A -85,B 0,C 180,E1 -5693.914,E2 -5693.914} C_VEL
LIN {X 0,Y 502.885,Z 408.845,A -85,B 0,C 180,E1 -5696.565,E2 -5696.565} C_VEL
LIN {X 0,Y 502.828,Z 408.853,A -85,B 0,C 180,E1 -5699.288,E2 -5699.288} C_VEL
LIN {X 0,Y 502.786,Z 408.856,A -85,B 0,C 180,E1 -5702.084,E2 -5702.084} C_VEL
LIN {X 0,Y 502.813,Z 408.856,A -85,B 0,C 180,E1 -5704.965,E2 -5704.965} C_VEL
LIN {X 0,Y 502.801,Z 408.855,A -85,B 0,C 180,E1 -5707.953,E2 -5707.953} C_VEL
LIN {X 0,Y 502.83,Z 408.853,A -85,B 0,C 180,E1 -5711.065,E2 -5711.065} C_VEL
LIN {X 0,Y 502.786,Z 408.858,A -85,B 0,C 180,E1 -5713.376,E2 -5713.376} C_VEL
LIN {X 0,Y 502.793,Z 408.855,A -85,B 0,C 180,E1 -5715.661,E2 -5715.661} C_VEL
LIN {X 0,Y 502.833,Z 408.85,A -85,B 0,C 180,E1 -5717.864,E2 -5717.864} C_VEL
LIN {X 0,Y 502.804,Z 408.856,A -85,B 0,C 180,E1 -5721.024,E2 -5721.024} C_VEL
LIN {X 0,Y 502.778,Z 408.859,A -85,B 0,C 180,E1 -5724.169,E2 -5724.169} C_VEL
LIN {X 0,Y 502.836,Z 408.853,A -85,B 0,C 180,E1 -5726.993,E2 -5726.993} C_VEL
LIN {X 0,Y 502.818,Z 408.852,A -85,B 0,C 180,E1 -5730.065,E2 -5730.065} C_VEL
LIN {X 0,Y 502.837,Z 408.853,A -85,B 0,C 180,E1 -5732.533,E2 -5732.533} C_VEL
LIN {X 0,Y 502.806,Z 408.856,A -85,B 0,C 180,E1 -5735.305,E2 -5735.305} C_VEL
LIN {X 0,Y 502.783,Z 408.858,A -85,B 0,C 180,E1 -5737.826,E2 -5737.826} C_VEL
LIN {X 0,Y 502.83,Z 408.852,A -85,B 0,C 180,E1 -5740.4,E2 -5740.4} C_VEL
LIN {X 0,Y 502.84,Z 408.853,A -85,B 0,C 180,E1 -5742.932,E2 -5742.932} C_VEL
LIN {X 0,Y 502.849,Z 408.848,A -85,B 0,C 180,E1 -5745.429,E2 -5745.429} C_VEL
LIN {X 0,Y 502.896,Z 408.844,A -85,B 0,C 180,E1 -5748.717,E2 -5748.717} C_VEL
LIN {X 0,Y 502.884,Z 408.845,A -85,B 0,C 180,E1 -5751.966,E2 -5751.966} C_VEL
LIN {X 0,Y 502.941,Z 408.839,A -85,B 0,C 180,E1 -5754.386,E2 -5754.386} C_VEL
LIN {X 0,Y 503.028,Z 408.826,A -85,B 0,C 180,E1 -5757.598,E2 -5757.598} C_VEL
LIN {X 0,Y 503.031,Z 408.828,A -85,B 0,C 180,E1 -5760,E2 -5760} C_VEL
LIN {X 0,Y 503.029,Z 408.828,A -85,B 0,C 180,E1 -5762.402,E2 -5762.402} C_VEL
LIN {X 0,Y 502.942,Z 408.838,A -85,B 0,C 180,E1 -5765.613,E2 -5765.613} C_VEL
LIN {X 0,Y 502.883,Z 408.846,A -85,B 0,C 180,E1 -5768.034,E2 -5768.034} C_VEL
LIN {X 0,Y 502.896,Z 408.843,A -85,B 0,C 180,E1 -5771.283,E2 -5771.283} C_VEL
LIN {X 0,Y 502.849,Z 408.851,A -85,B 0,C 180,E1 -5774.571,E2 -5774.571} C_VEL
LIN {X 0,Y 502.866,Z 408.849,A -85,B 0,C 180,E1 -5777.907,E2 -5777.907} C_VEL
LIN {X 0,Y 502.832,Z 408.852,A -85,B 0,C 180,E1 -5780.536,E2 -5780.536} C_VEL
LIN {X 0,Y 502.791,Z 408.856,A -85,B 0,C 180,E1 -5783.041,E2 -5783.041} C_VEL
LIN {X 0,Y 502.825,Z 408.854,A -85,B 0,C 180,E1 -5785.676,E2 -5785.676} C_VEL
LIN {X 0,Y 502.843,Z 408.852,A -85,B 0,C 180,E1 -5788.373,E2 -5788.373} C_VEL
LIN {X 0,Y 502.8,Z 408.855,A -85,B 0,C 180,E1 -5791.5,E2 -5791.5} C_VEL
LIN {X 0,Y 502.808,Z 408.855,A -85,B 0,C 180,E1 -5794.444,E2 -5794.444} C_VEL
LIN {X 0,Y 502.784,Z 408.858,A -85,B 0,C 180,E1 -5797.178,E2 -5797.178} C_VEL
LIN {X 0,Y 502.79,Z 408.858,A -85,B 0,C 180,E1 -5800.015,E2 -5800.015} C_VEL
LIN {X 0,Y 502.805,Z 408.857,A -85,B 0,C 180,E1 -5802.199,E2 -5802.199} C_VEL
LIN {X 0,Y 502.803,Z 408.857,A -85,B 0,C 180,E1 -5805.468,E2 -5805.468} C_VEL
LIN {X 0,Y 502.829,Z 408.851,A -85,B 0,C 180,E1 -5809.004,E2 -5809.004} C_VEL
LIN {X 0,Y 502.866,Z 409.042,A -85,B 0,C 180,E1 -5811.176,E2 -5811.176} C_VEL
LIN {X 0,Y 504.626,Z 418.316,A -85,B 0,C 180,E1 -5813.583,E2 -5813.583} C_VEL
LIN {X 0,Y 504.541,Z 425.433,A -85,B 0,C 180,E1 -5815.27,E2 -5815.27} C_VEL
LIN {X 0,Y 504.13,Z 440.125,A -85,B 0,C 180,E1 -5818.596,E2 -5818.596} C_VEL
LIN {X 0,Y 503.882,Z 453.401,A -85,B 0,C 180,E1 -5821.487,E2 -5821.487} C_VEL
LIN {X 0,Y 503.573,Z 468.99,A -85,B 0,C 180,E1 -5824.792,E2 -5824.792} C_VEL
LIN {X 0,Y 503.276,Z 483.595,A -85,B 0,C 180,E1 -5827.849,E2 -5827.849} C_VEL
LIN {X 0,Y 503.03,Z 497.944,A -85,B 0,C 180,E1 -5830.833,E2 -5830.833} C_VEL
LIN {X 0,Y 502.819,Z 511.202,A -85,B 0,C 180,E1 -5833.558,E2 -5833.558} C_VEL
LIN {X 0,Y 502.634,Z 521.473,A -85,B 0,C 180,E1 -5835.656,E2 -5835.656} C_VEL
LIN {X 0,Y 503.903,Z 532.779,A -85,B 0,C 180,E1 -5835.924,E2 -5835.924} C_VEL
LIN {X 0,Y 504.56,Z 539.115,A -85,B 0,C 180,E1 -5836.123,E2 -5836.123} C_VEL
LIN {X 0,Y 504.217,Z 551.777,A -85,B 0,C 180,E1 -5836.601,E2 -5836.601} C_VEL
LIN {X 0,Y 503.833,Z 564.765,A -85,B 0,C 180,E1 -5837.273,E2 -5837.273} C_VEL
LIN {X 0,Y 503.545,Z 575.788,A -85,B 0,C 180,E1 -5838.018,E2 -5838.018} C_VEL
LIN {X 0,Y 503.139,Z 586.612,A -85,B 0,C 180,E1 -5838.927,E2 -5838.927} C_VEL
LIN {X 0,Y 502.866,Z 596.402,A -85,B 0,C 180,E1 -5839.939,E2 -5839.939} C_VEL
LIN {X 0,Y 502.654,Z 604.447,A -85,B 0,C 180,E1 -5840.95,E2 -5840.95} C_VEL
LIN {X 0,Y 502.428,Z 612.318,A -85,B 0,C 180,E1 -5842.161,E2 -5842.161} C_VEL
LIN {X 0,Y 502.275,Z 619.586,A -85,B 0,C 180,E1 -5843.573,E2 -5843.573} C_VEL
LIN {X 0,Y 502.236,Z 624.437,A -85,B 0,C 180,E1 -5844.781,E2 -5844.781} C_VEL
LIN {X 0,Y 502.253,Z 628.153,A -85,B 0,C 180,E1 -5845.988,E2 -5845.988} C_VEL
LIN {X 0,Y 502.186,Z 630.061,A -85,B 0,C 180,E1 -5846.791,E2 -5846.791} C_VEL
LIN {X 0,Y 502.151,Z 631.494,A -85,B 0,C 180,E1 -5847.594,E2 -5847.594} C_VEL
LIN {X 0,Y 502.059,Z 633.132,A -85,B 0,C 180,E1 -5849.198,E2 -5849.198} C_VEL
LIN {X 0,Y 502.077,Z 633.358,A -85,B 0,C 180,E1 -5850,E2 -5850} C_VEL
LIN {X 0,Y 502.09,Z 632.512,A -85,B 0,C 180,E1 -5851.604,E2 -5851.604} C_VEL
LIN {X 0,Y 502.151,Z 631.497,A -85,B 0,C 180,E1 -5852.406,E2 -5852.406} C_VEL
LIN {X 0,Y 502.186,Z 630.064,A -85,B 0,C 180,E1 -5853.209,E2 -5853.209} C_VEL
LIN {X 0,Y 502.201,Z 627.046,A -85,B 0,C 180,E1 -5854.414,E2 -5854.414} C_VEL
LIN {X 0,Y 502.285,Z 622.971,A -85,B 0,C 180,E1 -5855.621,E2 -5855.621} C_VEL
LIN {X 0,Y 502.334,Z 616.799,A -85,B 0,C 180,E1 -5857.012,E2 -5857.012} C_VEL
LIN {X 0,Y 502.495,Z 609.864,A -85,B 0,C 180,E1 -5858.242,E2 -5858.242} C_VEL
LIN {X 0,Y 502.723,Z 601.405,A -85,B 0,C 180,E1 -5859.455,E2 -5859.455} C_VEL
LIN {X 0,Y 502.968,Z 592.747,A -85,B 0,C 180,E1 -5860.466,E2 -5860.466} C_VEL
LIN {X 0,Y 503.316,Z 582.083,A -85,B 0,C 180,E1 -5861.477,E2 -5861.477} C_VEL
LIN {X 0,Y 503.59,Z 570.862,A -85,B 0,C 180,E1 -5862.337,E2 -5862.337} C_VEL
LIN {X 0,Y 503.981,Z 560.044,A -85,B 0,C 180,E1 -5862.995,E2 -5862.995} C_VEL
LIN {X 0,Y 504.322,Z 548.259,A -85,B 0,C 180,E1 -5863.55,E2 -5863.55} C_VEL
LIN {X 0,Y 504.469,Z 536.543,A -85,B 0,C 180,E1 -5863.957,E2 -5863.957} C_VEL
LIN {X 0,Y 502.938,Z 524.89,A -85,B 0,C 180,E1 -5864.271,E2 -5864.271} C_VEL
LIN {X 0,Y 502.634,Z 521.46,A -85,B 0,C 180,E1 -5864.345,E2 -5864.345} C_VEL
LIN {X 0,Y 502.931,Z 506.11,A -85,B 0,C 180,E1 -5867.484,E2 -5867.484} C_VEL
LIN {X 0,Y 503.154,Z 490.877,A -85,B 0,C 180,E1 -5870.634,E2 -5870.634} C_VEL
LIN {X 0,Y 503.41,Z 476.359,A -85,B 0,C 180,E1 -5873.664,E2 -5873.664} C_VEL
LIN {X 0,Y 503.668,Z 462.762,A -85,B 0,C 180,E1 -5876.521,E2 -5876.521} C_VEL
LIN {X 0,Y 503.929,Z 449.074,A -85,B 0,C 180,E1 -5879.447,E2 -5879.447} C_VEL
LIN {X 0,Y 504.178,Z 436.458,A -85,B 0,C 180,E1 -5882.221,E2 -5882.221} C_VEL
LIN {X 0,Y 504.69,Z 421.912,A -85,B 0,C 180,E1 -5885.548,E2 -5885.548} C_VEL
LIN {X 0,Y 504.616,Z 418.297,A -85,B 0,C 180,E1 -5886.419,E2 -5886.419} C_VEL
LIN {X 0,Y 502.83,Z 408.851,A -85,B 0,C 180,E1 -5888.907,E2 -5888.907} C_VEL
LIN {X 0,Y 502.831,Z 408.854,A -85,B 0,C 180,E1 -5891.065,E2 -5891.065} C_VEL
LIN {X 0,Y 502.804,Z 408.858,A -85,B 0,C 180,E1 -5894.532,E2 -5894.532} C_VEL
LIN {X 0,Y 502.833,Z 408.853,A -85,B 0,C 180,E1 -5897.864,E2 -5897.864} C_VEL
LIN {X 0,Y 502.805,Z 408.854,A -85,B 0,C 180,E1 -5901.024,E2 -5901.024} C_VEL
LIN {X 0,Y 502.788,Z 408.859,A -85,B 0,C 180,E1 -5904.168,E2 -5904.168} C_VEL
LIN {X 0,Y 502.837,Z 408.851,A -85,B 0,C 180,E1 -5906.993,E2 -5906.993} C_VEL
LIN {X 0,Y 502.819,Z 408.854,A -85,B 0,C 180,E1 -5910.065,E2 -5910.065} C_VEL
LIN {X 0,Y 502.838,Z 408.851,A -85,B 0,C 180,E1 -5912.533,E2 -5912.533} C_VEL
LIN {X 0,Y 502.807,Z 408.854,A -85,B 0,C 180,E1 -5915.305,E2 -5915.305} C_VEL
LIN {X 0,Y 502.784,Z 408.86,A -85,B 0,C 180,E1 -5917.827,E2 -5917.827} C_VEL
LIN {X 0,Y 502.83,Z 408.852,A -85,B 0,C 180,E1 -5920.4,E2 -5920.4} C_VEL
LIN {X 0,Y 502.84,Z 408.85,A -85,B 0,C 180,E1 -5922.932,E2 -5922.932} C_VEL
LIN {X 0,Y 502.85,Z 408.851,A -85,B 0,C 180,E1 -5925.429,E2 -5925.429} C_VEL
LIN {X 0,Y 502.896,Z 408.842,A -85,B 0,C 180,E1 -5928.717,E2 -5928.717} C_VEL
LIN {X 0,Y 502.884,Z 408.846,A -85,B 0,C 180,E1 -5931.966,E2 -5931.966} C_VEL
LIN {X 0,Y 502.943,Z 408.838,A -85,B 0,C 180,E1 -5934.387,E2 -5934.387} C_VEL
LIN {X 0,Y 503.03,Z 408.828,A -85,B 0,C 180,E1 -5937.598,E2 -5937.598} C_VEL
LIN {X 0,Y 503.032,Z 408.828,A -85,B 0,C 180,E1 -5940,E2 -5940} C_VEL
LIN {X 0,Y 503.029,Z 408.826,A -85,B 0,C 180,E1 -5942.402,E2 -5942.402} C_VEL
LIN {X 0,Y 502.939,Z 408.839,A -85,B 0,C 180,E1 -5945.614,E2 -5945.614} C_VEL
LIN {X 0,Y 502.885,Z 408.845,A -85,B 0,C 180,E1 -5948.034,E2 -5948.034} C_VEL
LIN {X 0,Y 502.897,Z 408.844,A -85,B 0,C 180,E1 -5951.283,E2 -5951.283} C_VEL
LIN {X 0,Y 502.85,Z 408.848,A -85,B 0,C 180,E1 -5954.571,E2 -5954.571} C_VEL
LIN {X 0,Y 502.867,Z 408.849,A -85,B 0,C 180,E1 -5957.907,E2 -5957.907} C_VEL
LIN {X 0,Y 502.833,Z 408.851,A -85,B 0,C 180,E1 -5960.536,E2 -5960.536} C_VEL
LIN {X 0,Y 502.795,Z 408.857,A -85,B 0,C 180,E1 -5963.041,E2 -5963.041} C_VEL
LIN {X 0,Y 502.844,Z 408.85,A -85,B 0,C 180,E1 -5965.676,E2 -5965.676} C_VEL
LIN {X 0,Y 502.845,Z 408.849,A -85,B 0,C 180,E1 -5968.373,E2 -5968.373} C_VEL
LIN {X 0,Y 502.801,Z 408.856,A -85,B 0,C 180,E1 -5971.5,E2 -5971.5} C_VEL
LIN {X 0,Y 502.808,Z 408.854,A -85,B 0,C 180,E1 -5973.994,E2 -5973.994} C_VEL
LIN {X 0,Y 502.781,Z 408.86,A -85,B 0,C 180,E1 -5977.178,E2 -5977.178} C_VEL
LIN {X 0,Y 502.791,Z 408.856,A -85,B 0,C 180,E1 -5980.015,E2 -5980.015} C_VEL
LIN {X 0,Y 502.806,Z 408.854,A -85,B 0,C 180,E1 -5982.199,E2 -5982.199} C_VEL
LIN {X 0,Y 502.805,Z 408.857,A -85,B 0,C 180,E1 -5985.468,E2 -5985.468} C_VEL
LIN {X 0,Y 502.834,Z 408.851,A -85,B 0,C 180,E1 -5987.864,E2 -5987.864} C_VEL
LIN {X 0,Y 502.826,Z 408.854,A -85,B 0,C 180,E1 -5991.026,E2 -5991.026} C_VEL
LIN {X 0,Y 502.779,Z 408.858,A -85,B 0,C 180,E1 -5994.169,E2 -5994.169} C_VEL
LIN {X 0,Y 502.812,Z 408.853,A -85,B 0,C 180,E1 -5997.22,E2 -5997.22} C_VEL
LIN {X 0,Y 502.11,Z 408.94,A -85,B 0,C 180,E1 -5997.889,E2 -5997.889} C_VEL
LIN {X 0,Y 499.245,Z 409.299,A -85,B 0,C 180,E1 -5998.974,E2 -5998.974} C_VEL
LIN {X 0,Y 496.851,Z 409.596,A -85,B 0,C 180,E1 -5999.849,E2 -5999.849} C_VEL
LIN {X 0,Y 495.835,Z 409.724,A -85,B 0,C 180,E1 -6000.525,E2 -6000.525} C_VEL
LIN {X 0,Y 495.757,Z 409.731,A -85,B 0,C 180,E1 -6000.754,E2 -6000.754} C_VEL
LIN {X 0,Y 495.795,Z 409.728,A -85,B 0,C 180,E1 -6003.932,E2 -6003.932} C_VEL
LIN {X 0,Y 495.77,Z 409.732,A -85,B 0,C 180,E1 -6007.138,E2 -6007.138} C_VEL
LIN {X 0,Y 495.775,Z 409.731,A -85,B 0,C 180,E1 -6010.11,E2 -6010.11} C_VEL
LIN {X 0,Y 495.785,Z 409.73,A -85,B 0,C 180,E1 -6012.681,E2 -6012.681} C_VEL
LIN {X 0,Y 495.794,Z 409.729,A -85,B 0,C 180,E1 -6015.217,E2 -6015.217} C_VEL
LIN {X 0,Y 495.8,Z 409.729,A -85,B 0,C 180,E1 -6016.265,E2 -6016.265} C_VEL
LIN {X 0,Y 497.856,Z 417.729,A -85,B 0,C 180,E1 -6016.738,E2 -6016.738} C_VEL
LIN {X 0,Y 497.58,Z 428.588,A -85,B 0,C 180,E1 -6017.387,E2 -6017.387} C_VEL
LIN {X 0,Y 497.246,Z 439.055,A -85,B 0,C 180,E1 -6018.174,E2 -6018.174} C_VEL
LIN {X 0,Y 496.97,Z 447.903,A -85,B 0,C 180,E1 -6018.994,E2 -6018.994} C_VEL
LIN {X 0,Y 496.588,Z 456.976,A -85,B 0,C 180,E1 -6020.016,E2 -6020.016} C_VEL
LIN {X 0,Y 496.205,Z 465.757,A -85,B 0,C 180,E1 -6021.242,E2 -6021.242} C_VEL
LIN {X 0,Y 495.963,Z 472.805,A -85,B 0,C 180,E1 -6022.468,E2 -6022.468} C_VEL
LIN {X 0,Y 495.806,Z 477.555,A -85,B 0,C 180,E1 -6023.489,E2 -6023.489} C_VEL
LIN {X 0,Y 495.567,Z 482.178,A -85,B 0,C 180,E1 -6024.711,E2 -6024.711} C_VEL
LIN {X 0,Y 495.496,Z 485.699,A -85,B 0,C 180,E1 -6025.933,E2 -6025.933} C_VEL
LIN {X 0,Y 495.417,Z 487.524,A -85,B 0,C 180,E1 -6026.747,E2 -6026.747} C_VEL
LIN {X 0,Y 495.324,Z 488.906,A -85,B 0,C 180,E1 -6027.56,E2 -6027.56} C_VEL
LIN {X 0,Y 495.279,Z 490.483,A -85,B 0,C 180,E1 -6029.187,E2 -6029.187} C_VEL
LIN {X 0,Y 495.263,Z 490.716,A -85,B 0,C 180,E1 -6030,E2 -6030} C_VEL
LIN {X 0,Y 495.331,Z 489.96,A -85,B 0,C 180,E1 -6031.626,E2 -6031.626} C_VEL
LIN {X 0,Y 495.413,Z 487.695,A -85,B 0,C 180,E1 -6033.253,E2 -6033.253} C_VEL
LIN {X 0,Y 495.547,Z 484.891,A -85,B 0,C 180,E1 -6034.474,E2 -6034.474} C_VEL
LIN {X 0,Y 495.663,Z 481.095,A -85,B 0,C 180,E1 -6035.696,E2 -6035.696} C_VEL
LIN {X 0,Y 495.804,Z 475.185,A -85,B 0,C 180,E1 -6037.137,E2 -6037.137} C_VEL
LIN {X 0,Y 496.126,Z 468.799,A -85,B 0,C 180,E1 -6038.349,E2 -6038.349} C_VEL
LIN {X 0,Y 496.463,Z 460.785,A -85,B 0,C 180,E1 -6039.575,E2 -6039.575} C_VEL
LIN {X 0,Y 496.725,Z 452.576,A -85,B 0,C 180,E1 -6040.599,E2 -6040.599} C_VEL
LIN {X 0,Y 497.144,Z 442.397,A -85,B 0,C 180,E1 -6041.622,E2 -6041.622} C_VEL
LIN {X 0,Y 497.505,Z 431.936,A -85,B 0,C 180,E1 -6042.468,E2 -6042.468} C_VEL
LIN {X 0,Y 497.784,Z 421.246,A -85,B 0,C 180,E1 -6043.159,E2 -6043.159} C_VEL
LIN {X 0,Y 497.818,Z 417.481,A -85,B 0,C 180,E1 -6043.366,E2 -6043.366} C_VEL
LIN {X 0,Y 495.791,Z 409.724,A -85,B 0,C 180,E1 -6043.84,E2 -6043.84} C_VEL
LIN {X 0,Y 495.776,Z 409.73,A -85,B 0,C 180,E1 -6046.47,E2 -6046.47} C_VEL
LIN {X 0,Y 495.785,Z 409.731,A -85,B 0,C 180,E1 -6049.028,E2 -6049.028} C_VEL
LIN {X 0,Y 495.748,Z 409.734,A -85,B 0,C 180,E1 -6051.629,E2 -6051.629} C_VEL
LIN {X 0,Y 495.784,Z 409.73,A -85,B 0,C 180,E1 -6054.874,E2 -6054.874} C_VEL
LIN {X 0,Y 495.825,Z 409.725,A -85,B 0,C 180,E1 -6056.974,E2 -6056.974} C_VEL
LIN {X 0,Y 495.768,Z 409.73,A -85,B 0,C 180,E1 -6060.147,E2 -6060.147} C_VEL
LIN {X 0,Y 495.796,Z 409.729,A -85,B 0,C 180,E1 -6063.244,E2 -6063.244} C_VEL
LIN {X 0,Y 495.732,Z 409.735,A -85,B 0,C 180,E1 -6066.09,E2 -6066.09} C_VEL
LIN {X 0,Y 495.782,Z 409.73,A -85,B 0,C 180,E1 -6068.77,E2 -6068.77} C_VEL
LIN {X 0,Y 495.782,Z 409.729,A -85,B 0,C 180,E1 -6071.779,E2 -6071.779} C_VEL
LIN {X 0,Y 495.752,Z 409.735,A -85,B 0,C 180,E1 -6075.139,E2 -6075.139} C_VEL
LIN {X 0,Y 495.78,Z 409.729,A -85,B 0,C 180,E1 -6078.221,E2 -6078.221} C_VEL
LIN {X 0,Y 495.753,Z 409.734,A -85,B 0,C 180,E1 -6081.408,E2 -6081.408} C_VEL
LIN {X 0,Y 495.751,Z 409.734,A -85,B 0,C 180,E1 -6084.462,E2 -6084.462} C_VEL
LIN {X 0,Y 495.771,Z 409.73,A -85,B 0,C 180,E1 -6087.406,E2 -6087.406} C_VEL
LIN {X 0,Y 495.769,Z 409.731,A -85,B 0,C 180,E1 -6090.254,E2 -6090.254} C_VEL
LIN {X 0,Y 495.827,Z 409.726,A -85,B 0,C 180,E1 -6093.251,E2 -6093.251} C_VEL
LIN {X 0,Y 495.746,Z 409.736,A -85,B 0,C 180,E1 -6096.612,E2 -6096.612} C_VEL
LIN {X 0,Y 495.781,Z 409.729,A -85,B 0,C 180,E1 -6099.324,E2 -6099.324} C_VEL
LIN {X 0,Y 495.802,Z 409.726,A -85,B 0,C 180,E1 -6101.829,E2 -6101.829} C_VEL
LIN {X 0,Y 495.827,Z 409.725,A -85,B 0,C 180,E1 -6104.548,E2 -6104.548} C_VEL
LIN {X 0,Y 495.88,Z 409.717,A -85,B 0,C 180,E1 -6107.939,E2 -6107.939} C_VEL
LIN {X 0,Y 495.84,Z 409.723,A -85,B 0,C 180,E1 -6111.03,E2 -6111.03} C_VEL
LIN {X 0,Y 495.883,Z 409.717,A -85,B 0,C 180,E1 -6113.49,E2 -6113.49} C_VEL
LIN {X 0,Y 495.847,Z 409.723,A -85,B 0,C 180,E1 -6116.75,E2 -6116.75} C_VEL
LIN {X 0,Y 496.009,Z 409.7,A -85,B 0,C 180,E1 -6119.188,E2 -6119.188} C_VEL
LIN {X 0,Y 495.876,Z 409.717,A -85,B 0,C 180,E1 -6121.624,E2 -6121.624} C_VEL
LIN {X 0,Y 495.849,Z 409.721,A -85,B 0,C 180,E1 -6123.25,E2 -6123.25} C_VEL
LIN {X 0,Y 495.883,Z 409.718,A -85,B 0,C 180,E1 -6126.51,E2 -6126.51} C_VEL
LIN {X 0,Y 495.837,Z 409.722,A -85,B 0,C 180,E1 -6128.97,E2 -6128.97} C_VEL
LIN {X 0,Y 495.855,Z 409.722,A -85,B 0,C 180,E1 -6132.275,E2 -6132.275} C_VEL
LIN {X 0,Y 495.811,Z 409.725,A -85,B 0,C 180,E1 -6135.624,E2 -6135.624} C_VEL
LIN {X 0,Y 495.81,Z 409.727,A -85,B 0,C 180,E1 -6138.247,E2 -6138.247} C_VEL
LIN {X 0,Y 495.777,Z 409.731,A -85,B 0,C 180,E1 -6140.756,E2 -6140.756} C_VEL
LIN {X 0,Y 495.745,Z 409.734,A -85,B 0,C 180,E1 -6143.387,E2 -6143.387} C_VEL
LIN {X 0,Y 495.826,Z 409.723,A -85,B 0,C 180,E1 -6146.749,E2 -6146.749} C_VEL
LIN {X 0,Y 495.769,Z 409.733,A -85,B 0,C 180,E1 -6149.746,E2 -6149.746} C_VEL
LIN {X 0,Y 495.772,Z 409.732,A -85,B 0,C 180,E1 -6152.594,E2 -6152.594} C_VEL
LIN {X 0,Y 495.759,Z 409.733,A -85,B 0,C 180,E1 -6155.537,E2 -6155.537} C_VEL
LIN {X 0,Y 495.766,Z 409.731,A -85,B 0,C 180,E1 -6158.768,E2 -6158.768} C_VEL
LIN {X 0,Y 495.78,Z 409.731,A -85,B 0,C 180,E1 -6161.779,E2 -6161.779} C_VEL
LIN {X 0,Y 495.752,Z 409.736,A -85,B 0,C 180,E1 -6165.139,E2 -6165.139} C_VEL
LIN {X 0,Y 495.763,Z 409.733,A -85,B 0,C 180,E1 -6168.219,E2 -6168.219} C_VEL
LIN {X 0,Y 495.819,Z 409.791,A -85,B 0,C 180,E1 -6170.884,E2 -6170.884} C_VEL
LIN {X 0,Y 497.744,Z 420.194,A -85,B 0,C 180,E1 -6173.628,E2 -6173.628} C_VEL
LIN {X 0,Y 497.509,Z 428.443,A -85,B 0,C 180,E1 -6175.594,E2 -6175.594} C_VEL
LIN {X 0,Y 497.137,Z 443.048,A -85,B 0,C 180,E1 -6178.936,E2 -6178.936} C_VEL
LIN {X 0,Y 496.793,Z 457.755,A -85,B 0,C 180,E1 -6182.17,E2 -6182.17} C_VEL
LIN {X 0,Y 496.463,Z 472.595,A -85,B 0,C 180,E1 -6185.354,E2 -6185.354} C_VEL
LIN {X 0,Y 496.186,Z 485.897,A -85,B 0,C 180,E1 -6188.173,E2 -6188.173} C_VEL
LIN {X 0,Y 495.947,Z 500.292,A -85,B 0,C 180,E1 -6191.214,E2 -6191.214} C_VEL
LIN {X 0,Y 495.701,Z 513.318,A -85,B 0,C 180,E1 -6193.95,E2 -6193.95} C_VEL
LIN {X 0,Y 495.582,Z 520.5,A -85,B 0,C 180,E1 -6195.447,E2 -6195.447} C_VEL
LIN {X 0,Y 496.951,Z 533.601,A -85,B 0,C 180,E1 -6195.776,E2 -6195.776} C_VEL
LIN {X 0,Y 497.617,Z 538.861,A -85,B 0,C 180,E1 -6195.951,E2 -6195.951} C_VEL
LIN {X 0,Y 497.244,Z 551.896,A -85,B 0,C 180,E1 -6196.462,E2 -6196.462} C_VEL
LIN {X 0,Y 496.858,Z 564.137,A -85,B 0,C 180,E1 -6197.116,E2 -6197.116} C_VEL
LIN {X 0,Y 496.49,Z 576.074,A -85,B 0,C 180,E1 -6197.948,E2 -6197.948} C_VEL
LIN {X 0,Y 496.057,Z 586.674,A -85,B 0,C 180,E1 -6198.87,E2 -6198.87} C_VEL
LIN {X 0,Y 495.798,Z 595.375,A -85,B 0,C 180,E1 -6199.794,E2 -6199.794} C_VEL
LIN {X 0,Y 495.58,Z 603.422,A -85,B 0,C 180,E1 -6200.82,E2 -6200.82} C_VEL
LIN {X 0,Y 495.37,Z 611.299,A -85,B 0,C 180,E1 -6202.049,E2 -6202.049} C_VEL
LIN {X 0,Y 495.204,Z 618.568,A -85,B 0,C 180,E1 -6203.481,E2 -6203.481} C_VEL
LIN {X 0,Y 495.196,Z 623.426,A -85,B 0,C 180,E1 -6204.707,E2 -6204.707} C_VEL
LIN {X 0,Y 495.197,Z 627.142,A -85,B 0,C 180,E1 -6205.931,E2 -6205.931} C_VEL
LIN {X 0,Y 495.143,Z 629.051,A -85,B 0,C 180,E1 -6206.745,E2 -6206.745} C_VEL
LIN {X 0,Y 495.112,Z 630.486,A -85,B 0,C 180,E1 -6207.559,E2 -6207.559} C_VEL
LIN {X 0,Y 495.057,Z 631.505,A -85,B 0,C 180,E1 -6208.373,E2 -6208.373} C_VEL
LIN {X 0,Y 495.069,Z 632.355,A -85,B 0,C 180,E1 -6210,E2 -6210} C_VEL
LIN {X 0,Y 495.057,Z 631.506,A -85,B 0,C 180,E1 -6211.627,E2 -6211.627} C_VEL
LIN {X 0,Y 495.112,Z 630.489,A -85,B 0,C 180,E1 -6212.441,E2 -6212.441} C_VEL
LIN {X 0,Y 495.143,Z 629.055,A -85,B 0,C 180,E1 -6213.255,E2 -6213.255} C_VEL
LIN {X 0,Y 495.144,Z 626.034,A -85,B 0,C 180,E1 -6214.478,E2 -6214.478} C_VEL
LIN {X 0,Y 495.266,Z 620.754,A -85,B 0,C 180,E1 -6216.004,E2 -6216.004} C_VEL
LIN {X 0,Y 495.277,Z 614.639,A -85,B 0,C 180,E1 -6217.337,E2 -6217.337} C_VEL
LIN {X 0,Y 495.471,Z 607.58,A -85,B 0,C 180,E1 -6218.565,E2 -6218.565} C_VEL
LIN {X 0,Y 495.685,Z 598.754,A -85,B 0,C 180,E1 -6219.796,E2 -6219.796} C_VEL
LIN {X 0,Y 496.004,Z 589.739,A -85,B 0,C 180,E1 -6220.821,E2 -6220.821} C_VEL
LIN {X 0,Y 496.409,Z 578.673,A -85,B 0,C 180,E1 -6221.846,E2 -6221.846} C_VEL
LIN {X 0,Y 496.731,Z 568.161,A -85,B 0,C 180,E1 -6222.627,E2 -6222.627} C_VEL
LIN {X 0,Y 497.062,Z 556.061,A -85,B 0,C 180,E1 -6223.335,E2 -6223.335} C_VEL
LIN {X 0,Y 497.485,Z 543.305,A -85,B 0,C 180,E1 -6223.896,E2 -6223.896} C_VEL
LIN {X 0,Y 497.409,Z 536.424,A -85,B 0,C 180,E1 -6224.133,E2 -6224.133} C_VEL
LIN {X 0,Y 496.091,Z 525.994,A -85,B 0,C 180,E1 -6224.433,E2 -6224.433} C_VEL
LIN {X 0,Y 495.569,Z 520.289,A -85,B 0,C 180,E1 -6224.58,E2 -6224.58} C_VEL
LIN {X 0,Y 495.838,Z 505.242,A -85,B 0,C 180,E1 -6227.743,E2 -6227.743} C_VEL
LIN {X 0,Y 496.103,Z 490.869,A -85,B 0,C 180,E1 -6230.774,E2 -6230.774} C_VEL
LIN {X 0,Y 496.41,Z 475.544,A -85,B 0,C 180,E1 -6234.019,E2 -6234.019} C_VEL
LIN {X 0,Y 496.671,Z 461.867,A -85,B 0,C 180,E1 -6236.942,E2 -6236.942} C_VEL
LIN {X 0,Y 496.94,Z 449.336,A -85,B 0,C 180,E1 -6239.669,E2 -6239.669} C_VEL
LIN {X 0,Y 497.206,Z 438.043,A -85,B 0,C 180,E1 -6242.194,E2 -6242.194} C_VEL
LIN {X 0,Y 497.766,Z 423.272,A -85,B 0,C 180,E1 -6245.621,E2 -6245.621} C_VEL
LIN {X 0,Y 497.717,Z 420.069,A -85,B 0,C 180,E1 -6246.402,E2 -6246.402} C_VEL
LIN {X 0,Y 495.8,Z 409.727,A -85,B 0,C 180,E1 -6249.132,E2 -6249.132} C_VEL
LIN {X 0,Y 495.764,Z 409.73,A -85,B 0,C 180,E1 -6251.781,E2 -6251.781} C_VEL
LIN {X 0,Y 495.753,Z 409.734,A -85,B 0,C 180,E1 -6255.139,E2 -6255.139} C_VEL
LIN {X 0,Y 495.781,Z 409.731,A -85,B 0,C 180,E1 -6258.221,E2 -6258.221} C_VEL
LIN {X 0,Y 495.754,Z 409.732,A -85,B 0,C 180,E1 -6261.409,E2 -6261.409} C_VEL
LIN {X 0,Y 495.76,Z 409.733,A -85,B 0,C 180,E1 -6264.463,E2 -6264.463} C_VEL
LIN {X 0,Y 495.773,Z 409.731,A -85,B 0,C 180,E1 -6267.406,E2 -6267.406} C_VEL
LIN {X 0,Y 495.77,Z 409.733,A -85,B 0,C 180,E1 -6270.254,E2 -6270.254} C_VEL
LIN {X 0,Y 495.827,Z 409.723,A -85,B 0,C 180,E1 -6273.251,E2 -6273.251} C_VEL
LIN {X 0,Y 495.746,Z 409.734,A -85,B 0,C 180,E1 -6276.613,E2 -6276.613} C_VEL
LIN {X 0,Y 495.782,Z 409.73,A -85,B 0,C 180,E1 -6279.324,E2 -6279.324} C_VEL
LIN {X 0,Y 495.803,Z 409.728,A -85,B 0,C 180,E1 -6281.829,E2 -6281.829} C_VEL
LIN {X 0,Y 495.828,Z 409.723,A -85,B 0,C 180,E1 -6284.548,E2 -6284.548} C_VEL
LIN {X 0,Y 495.881,Z 409.718,A -85,B 0,C 180,E1 -6287.939,E2 -6287.939} C_VEL
LIN {X 0,Y 495.838,Z 409.722,A -85,B 0,C 180,E1 -6291.03,E2 -6291.03} C_VEL
LIN {X 0,Y 495.884,Z 409.718,A -85,B 0,C 180,E1 -6293.49,E2 -6293.49} C_VEL
LIN {X 0,Y 495.849,Z 409.721,A -85,B 0,C 180,E1 -6296.75,E2 -6296.75} C_VEL
LIN {X 0,Y 496.01,Z 409.703,A -85,B 0,C 180,E1 -6299.188,E2 -6299.188} C_VEL
LIN {X 0,Y 495.876,Z 409.719,A -85,B 0,C 180,E1 -6301.624,E2 -6301.624} C_VEL
LIN {X 0,Y 495.848,Z 409.723,A -85,B 0,C 180,E1 -6303.25,E2 -6303.25} C_VEL
LIN {X 0,Y 495.869,Z 409.718,A -85,B 0,C 180,E1 -6306.511,E2 -6306.511} C_VEL
LIN {X 0,Y 495.842,Z 409.723,A -85,B 0,C 180,E1 -6308.97,E2 -6308.97} C_VEL
LIN {X 0,Y 495.856,Z 409.719,A -85,B 0,C 180,E1 -6312.275,E2 -6312.275} C_VEL
LIN {X 0,Y 495.812,Z 409.727,A -85,B 0,C 180,E1 -6315.624,E2 -6315.624} C_VEL
LIN {X 0,Y 495.811,Z 409.725,A -85,B 0,C 180,E1 -6318.247,E2 -6318.247} C_VEL
LIN {X 0,Y 495.778,Z 409.73,A -85,B 0,C 180,E1 -6320.756,E2 -6320.756} C_VEL
LIN {X 0,Y 495.751,Z 409.736,A -85,B 0,C 180,E1 -6323.387,E2 -6323.387} C_VEL
LIN {X 0,Y 495.795,Z 409.727,A -85,B 0,C 180,E1 -6326.068,E2 -6326.068} C_VEL
LIN {X 0,Y 495.776,Z 409.732,A -85,B 0,C 180,E1 -6328.815,E2 -6328.815} C_VEL
LIN {X 0,Y 495.763,Z 409.733,A -85,B 0,C 180,E1 -6331.726,E2 -6331.726} C_VEL
LIN {X 0,Y 495.773,Z 409.731,A -85,B 0,C 180,E1 -6334.694,E2 -6334.694} C_VEL
LIN {X 0,Y 495.732,Z 409.736,A -85,B 0,C 180,E1 -6337.562,E2 -6337.562} C_VEL
LIN {X 0,Y 495.77,Z 409.732,A -85,B 0,C 180,E1 -6340.7,E2 -6340.7} C_VEL
LIN {X 0,Y 495.739,Z 409.734,A -85,B 0,C 180,E1 -6343.695,E2 -6343.695} C_VEL
LIN {X 0,Y 495.739,Z 409.734,A -85,B 0,C 180,E1 -6346.305,E2 -6346.305} C_VEL
LIN {X 0,Y 495.785,Z 409.73,A -85,B 0,C 180,E1 -6349.302,E2 -6349.302} C_VEL
LIN {X 0,Y 495.768,Z 409.732,A -85,B 0,C 180,E1 -6351.41,E2 -6351.41} C_VEL
LIN {X 0,Y 495.752,Z 409.734,A -85,B 0,C 180,E1 -6354.462,E2 -6354.462} C_VEL
LIN {X 0,Y 495.771,Z 409.731,A -85,B 0,C 180,E1 -6357.406,E2 -6357.406} C_VEL
LIN {X 0,Y 495.757,Z 409.731,A -85,B 0,C 180,E1 -6360.754,E2 -6360.754} C_VEL
LIN {X 0,Y 495.1,Z 409.816,A -85,B 0,C 180,E1 -6361.433,E2 -6361.433} C_VEL
LIN {X 0,Y 492.244,Z 410.171,A -85,B 0,C 180,E1 -6362.535,E2 -6362.535} C_VEL
LIN {X 0,Y 489.835,Z 410.471,A -85,B 0,C 180,E1 -6363.424,E2 -6363.424} C_VEL
LIN {X 0,Y 488.819,Z 410.597,A -85,B 0,C 180,E1 -6364.11,E2 -6364.11} C_VEL
LIN {X 0,Y 488.747,Z 410.605,A -85,B 0,C 180,E1 -6364.343,E2 -6364.343} C_VEL
LIN {X 0,Y 488.732,Z 410.608,A -85,B 0,C 180,E1 -6367.153,E2 -6367.153} C_VEL
LIN {X 0,Y 488.729,Z 410.607,A -85,B 0,C 180,E1 -6369.81,E2 -6369.81} C_VEL
LIN {X 0,Y 488.733,Z 410.609,A -85,B 0,C 180,E1 -6372.423,E2 -6372.423} C_VEL
LIN {X 0,Y 488.766,Z 410.604,A -85,B 0,C 180,E1 -6375,E2 -6375} C_VEL
LIN {X 0,Y 488.757,Z 410.606,A -85,B 0,C 180,E1 -6376.063,E2 -6376.063} C_VEL
LIN {X 0,Y 490.973,Z 418.751,A -85,B 0,C 180,E1 -6376.549,E2 -6376.549} C_VEL
LIN {X 0,Y 490.727,Z 429.603,A -85,B 0,C 180,E1 -6377.208,E2 -6377.208} C_VEL
LIN {X 0,Y 490.371,Z 440.067,A -85,B 0,C 180,E1 -6378.006,E2 -6378.006} C_VEL
LIN {X 0,Y 490.078,Z 448.913,A -85,B 0,C 180,E1 -6378.837,E2 -6378.837} C_VEL
LIN {X 0,Y 489.677,Z 457.984,A -85,B 0,C 180,E1 -6379.874,E2 -6379.874} C_VEL
LIN {X 0,Y 489.266,Z 466.765,A -85,B 0,C 180,E1 -6381.117,E2 -6381.117} C_VEL
LIN {X 0,Y 488.997,Z 473.814,A -85,B 0,C 180,E1 -6382.36,E2 -6382.36} C_VEL
LIN {X 0,Y 488.83,Z 478.562,A -85,B 0,C 180,E1 -6383.395,E2 -6383.395} C_VEL
LIN {X 0,Y 488.574,Z 483.184,A -85,B 0,C 180,E1 -6384.635,E2 -6384.635} C_VEL
LIN {X 0,Y 488.486,Z 486.706,A -85,B 0,C 180,E1 -6385.875,E2 -6385.875} C_VEL
LIN {X 0,Y 488.4,Z 488.531,A -85,B 0,C 180,E1 -6386.7,E2 -6386.7} C_VEL
LIN {X 0,Y 488.303,Z 489.912,A -85,B 0,C 180,E1 -6387.525,E2 -6387.525} C_VEL
LIN {X 0,Y 488.257,Z 491.487,A -85,B 0,C 180,E1 -6389.175,E2 -6389.175} C_VEL
LIN {X 0,Y 488.239,Z 491.72,A -85,B 0,C 180,E1 -6390,E2 -6390} C_VEL
LIN {X 0,Y 488.315,Z 490.963,A -85,B 0,C 180,E1 -6391.649,E2 -6391.649} C_VEL
LIN {X 0,Y 488.396,Z 488.699,A -85,B 0,C 180,E1 -6393.3,E2 -6393.3} C_VEL
LIN {X 0,Y 488.541,Z 485.894,A -85,B 0,C 180,E1 -6394.538,E2 -6394.538} C_VEL
LIN {X 0,Y 488.678,Z 482.096,A -85,B 0,C 180,E1 -6395.778,E2 -6395.778} C_VEL
LIN {X 0,Y 488.831,Z 476.191,A -85,B 0,C 180,E1 -6397.239,E2 -6397.239} C_VEL
LIN {X 0,Y 489.176,Z 469.8,A -85,B 0,C 180,E1 -6398.468,E2 -6398.468} C_VEL
LIN {X 0,Y 489.547,Z 461.784,A -85,B 0,C 180,E1 -6399.711,E2 -6399.711} C_VEL
LIN {X 0,Y 489.825,Z 453.575,A -85,B 0,C 180,E1 -6400.75,E2 -6400.75} C_VEL
LIN {X 0,Y 490.263,Z 443.395,A -85,B 0,C 180,E1 -6401.787,E2 -6401.787} C_VEL
LIN {X 0,Y 490.644,Z 432.946,A -85,B 0,C 180,E1 -6402.644,E2 -6402.644} C_VEL
LIN {X 0,Y 490.942,Z 422.241,A -85,B 0,C 180,E1 -6403.346,E2 -6403.346} C_VEL
LIN {X 0,Y 490.925,Z 418.484,A -85,B 0,C 180,E1 -6403.558,E2 -6403.558} C_VEL
LIN {X 0,Y 488.767,Z 410.597,A -85,B 0,C 180,E1 -6404.043,E2 -6404.043} C_VEL
LIN {X 0,Y 488.724,Z 410.609,A -85,B 0,C 180,E1 -6406.715,E2 -6406.715} C_VEL
LIN {X 0,Y 488.746,Z 410.607,A -85,B 0,C 180,E1 -6409.313,E2 -6409.313} C_VEL
LIN {X 0,Y 488.705,Z 410.612,A -85,B 0,C 180,E1 -6411.957,E2 -6411.957} C_VEL
LIN {X 0,Y 488.75,Z 410.606,A -85,B 0,C 180,E1 -6415.053,E2 -6415.053} C_VEL
LIN {X 0,Y 488.754,Z 410.608,A -85,B 0,C 180,E1 -6417.396,E2 -6417.396} C_VEL
LIN {X 0,Y 488.713,Z 410.609,A -85,B 0,C 180,E1 -6420.363,E2 -6420.363} C_VEL
LIN {X 0,Y 488.739,Z 410.608,A -85,B 0,C 180,E1 -6423.484,E2 -6423.484} C_VEL
LIN {X 0,Y 488.692,Z 410.612,A -85,B 0,C 180,E1 -6426.356,E2 -6426.356} C_VEL
LIN {X 0,Y 488.752,Z 410.607,A -85,B 0,C 180,E1 -6429.249,E2 -6429.249} C_VEL
LIN {X 0,Y 488.739,Z 410.608,A -85,B 0,C 180,E1 -6432.521,E2 -6432.521} C_VEL
LIN {X 0,Y 488.705,Z 410.609,A -85,B 0,C 180,E1 -6435.976,E2 -6435.976} C_VEL
LIN {X 0,Y 488.722,Z 410.61,A -85,B 0,C 180,E1 -6438.586,E2 -6438.586} C_VEL
LIN {X 0,Y 488.682,Z 410.613,A -85,B 0,C 180,E1 -6441.8,E2 -6441.8} C_VEL
LIN {X 0,Y 488.726,Z 410.61,A -85,B 0,C 180,E1 -6445.052,E2 -6445.052} C_VEL
LIN {X 0,Y 488.707,Z 410.61,A -85,B 0,C 180,E1 -6448.046,E2 -6448.046} C_VEL
LIN {X 0,Y 488.727,Z 410.61,A -85,B 0,C 180,E1 -6450.73,E2 -6450.73} C_VEL
LIN {X 0,Y 488.756,Z 410.604,A -85,B 0,C 180,E1 -6453.528,E2 -6453.528} C_VEL
LIN {X 0,Y 488.682,Z 410.614,A -85,B 0,C 180,E1 -6456.254,E2 -6456.254} C_VEL
LIN {X 0,Y 488.749,Z 410.606,A -85,B 0,C 180,E1 -6459.176,E2 -6459.176} C_VEL
LIN {X 0,Y 488.763,Z 410.603,A -85,B 0,C 180,E1 -6461.628,E2 -6461.628} C_VEL
LIN {X 0,Y 488.766,Z 410.605,A -85,B 0,C 180,E1 -6465,E2 -6465} C_VEL
LIN {X 0,Y 488.833,Z 410.598,A -85,B 0,C 180,E1 -6468.388,E2 -6468.388} C_VEL
LIN {X 0,Y 488.789,Z 410.6,A -85,B 0,C 180,E1 -6471.733,E2 -6471.733} C_VEL
LIN {X 0,Y 488.858,Z 410.593,A -85,B 0,C 180,E1 -6474.224,E2 -6474.224} C_VEL
LIN {X 0,Y 488.964,Z 410.577,A -85,B 0,C 180,E1 -6477.529,E2 -6477.529} C_VEL
LIN {X 0,Y 488.959,Z 410.581,A -85,B 0,C 180,E1 -6480.824,E2 -6480.824} C_VEL
LIN {X 0,Y 488.966,Z 410.58,A -85,B 0,C 180,E1 -6482.471,E2 -6482.471} C_VEL
LIN {X 0,Y 488.859,Z 410.592,A -85,B 0,C 180,E1 -6485.776,E2 -6485.776} C_VEL
LIN {X 0,Y 488.788,Z 410.602,A -85,B 0,C 180,E1 -6488.267,E2 -6488.267} C_VEL
LIN {X 0,Y 488.833,Z 410.595,A -85,B 0,C 180,E1 -6491.612,E2 -6491.612} C_VEL
LIN {X 0,Y 488.765,Z 410.602,A -85,B 0,C 180,E1 -6495,E2 -6495} C_VEL
LIN {X 0,Y 488.758,Z 410.605,A -85,B 0,C 180,E1 -6498.442,E2 -6498.442} C_VEL
LIN {X 0,Y 488.71,Z 410.61,A -85,B 0,C 180,E1 -6501.071,E2 -6501.071} C_VEL
LIN {X 0,Y 488.682,Z 410.615,A -85,B 0,C 180,E1 -6503.746,E2 -6503.746} C_VEL
LIN {X 0,Y 488.795,Z 410.598,A -85,B 0,C 180,E1 -6506.944,E2 -6506.944} C_VEL
LIN {X 0,Y 488.713,Z 410.611,A -85,B 0,C 180,E1 -6510.363,E2 -6510.363} C_VEL
LIN {X 0,Y 488.738,Z 410.607,A -85,B 0,C 180,E1 -6513.484,E2 -6513.484} C_VEL
LIN {X 0,Y 488.691,Z 410.613,A -85,B 0,C 180,E1 -6516.356,E2 -6516.356} C_VEL
LIN {X 0,Y 488.703,Z 410.612,A -85,B 0,C 180,E1 -6519.254,E2 -6519.254} C_VEL
LIN {X 0,Y 488.726,Z 410.61,A -85,B 0,C 180,E1 -6521.602,E2 -6521.602} C_VEL
LIN {X 0,Y 488.715,Z 410.613,A -85,B 0,C 180,E1 -6524.801,E2 -6524.801} C_VEL
LIN {X 0,Y 488.694,Z 410.613,A -85,B 0,C 180,E1 -6527.475,E2 -6527.475} C_VEL
LIN {X 0,Y 488.776,Z 410.681,A -85,B 0,C 180,E1 -6530.62,E2 -6530.62} C_VEL
LIN {X 0,Y 490.688,Z 420.727,A -85,B 0,C 180,E1 -6533.329,E2 -6533.329} C_VEL
LIN {X 0,Y 490.798,Z 425.185,A -85,B 0,C 180,E1 -6534.434,E2 -6534.434} C_VEL
LIN {X 0,Y 490.234,Z 440.19,A -85,B 0,C 180,E1 -6537.965,E2 -6537.965} C_VEL
LIN {X 0,Y 489.879,Z 452.747,A -85,B 0,C 180,E1 -6540.805,E2 -6540.805} C_VEL
LIN {X 0,Y 489.573,Z 466.37,A -85,B 0,C 180,E1 -6543.805,E2 -6543.805} C_VEL
LIN {X 0,Y 489.237,Z 481.965,A -85,B 0,C 180,E1 -6547.179,E2 -6547.179} C_VEL
LIN {X 0,Y 488.935,Z 496.31,A -85,B 0,C 180,E1 -6550.258,E2 -6550.258} C_VEL
LIN {X 0,Y 488.635,Z 510.4,A -85,B 0,C 180,E1 -6553.282,E2 -6553.282} C_VEL
LIN {X 0,Y 488.515,Z 519.533,A -85,B 0,C 180,E1 -6555.232,E2 -6555.232} C_VEL
LIN {X 0,Y 489.94,Z 533.951,A -85,B 0,C 180,E1 -6555.607,E2 -6555.607} C_VEL
LIN {X 0,Y 490.605,Z 540.137,A -85,B 0,C 180,E1 -6555.826,E2 -6555.826} C_VEL
LIN {X 0,Y 490.247,Z 553.049,A -85,B 0,C 180,E1 -6556.371,E2 -6556.371} C_VEL
LIN {X 0,Y 489.775,Z 565.369,A -85,B 0,C 180,E1 -6557.075,E2 -6557.075} C_VEL
LIN {X 0,Y 489.436,Z 576.361,A -85,B 0,C 180,E1 -6557.877,E2 -6557.877} C_VEL
LIN {X 0,Y 488.976,Z 586.714,A -85,B 0,C 180,E1 -6558.812,E2 -6558.812} C_VEL
LIN {X 0,Y 488.714,Z 596.071,A -85,B 0,C 180,E1 -6559.854,E2 -6559.854} C_VEL
LIN {X 0,Y 488.436,Z 605.201,A -85,B 0,C 180,E1 -6561.102,E2 -6561.102} C_VEL
LIN {X 0,Y 488.243,Z 612.568,A -85,B 0,C 180,E1 -6562.348,E2 -6562.348} C_VEL
LIN {X 0,Y 488.156,Z 618.842,A -85,B 0,C 180,E1 -6563.687,E2 -6563.687} C_VEL
LIN {X 0,Y 488.121,Z 623.763,A -85,B 0,C 180,E1 -6565.044,E2 -6565.044} C_VEL
LIN {X 0,Y 488.143,Z 626.13,A -85,B 0,C 180,E1 -6565.872,E2 -6565.872} C_VEL
LIN {X 0,Y 488.097,Z 628.042,A -85,B 0,C 180,E1 -6566.698,E2 -6566.698} C_VEL
LIN {X 0,Y 488.072,Z 629.478,A -85,B 0,C 180,E1 -6567.524,E2 -6567.524} C_VEL
LIN {X 0,Y 488.025,Z 630.498,A -85,B 0,C 180,E1 -6568.35,E2 -6568.35} C_VEL
LIN {X 0,Y 488.059,Z 631.353,A -85,B 0,C 180,E1 -6570,E2 -6570} C_VEL
LIN {X 0,Y 488.025,Z 630.5,A -85,B 0,C 180,E1 -6571.651,E2 -6571.651} C_VEL
LIN {X 0,Y 488.072,Z 629.481,A -85,B 0,C 180,E1 -6572.476,E2 -6572.476} C_VEL
LIN {X 0,Y 488.097,Z 628.046,A -85,B 0,C 180,E1 -6573.302,E2 -6573.302} C_VEL
LIN {X 0,Y 488.094,Z 625.022,A -85,B 0,C 180,E1 -6574.542,E2 -6574.542} C_VEL
LIN {X 0,Y 488.203,Z 619.91,A -85,B 0,C 180,E1 -6576.048,E2 -6576.048} C_VEL
LIN {X 0,Y 488.237,Z 613.624,A -85,B 0,C 180,E1 -6577.444,E2 -6577.444} C_VEL
LIN {X 0,Y 488.402,Z 606.557,A -85,B 0,C 180,E1 -6578.69,E2 -6578.69} C_VEL
LIN {X 0,Y 488.634,Z 597.731,A -85,B 0,C 180,E1 -6579.939,E2 -6579.939} C_VEL
LIN {X 0,Y 488.993,Z 587.719,A -85,B 0,C 180,E1 -6581.083,E2 -6581.083} C_VEL
LIN {X 0,Y 489.404,Z 577.668,A -85,B 0,C 180,E1 -6582.017,E2 -6582.017} C_VEL
LIN {X 0,Y 489.74,Z 567.137,A -85,B 0,C 180,E1 -6582.81,E2 -6582.81} C_VEL
LIN {X 0,Y 490.131,Z 555.042,A -85,B 0,C 180,E1 -6583.527,E2 -6583.527} C_VEL
LIN {X 0,Y 490.558,Z 542.284,A -85,B 0,C 180,E1 -6584.096,E2 -6584.096} C_VEL
LIN {X 0,Y 490.41,Z 537.016,A -85,B 0,C 180,E1 -6584.286,E2 -6584.286} C_VEL
LIN {X 0,Y 489.136,Z 526.114,A -85,B 0,C 180,E1 -6584.616,E2 -6584.616} C_VEL
LIN {X 0,Y 488.515,Z 519.453,A -85,B 0,C 180,E1 -6584.768,E2 -6584.768} C_VEL
LIN {X 0,Y 488.779,Z 504.517,A -85,B 0,C 180,E1 -6587.98,E2 -6587.98} C_VEL
LIN {X 0,Y 489.083,Z 489.163,A -85,B 0,C 180,E1 -6591.275,E2 -6591.275} C_VEL
LIN {X 0,Y 489.357,Z 475.749,A -85,B 0,C 180,E1 -6594.162,E2 -6594.162} C_VEL
LIN {X 0,Y 489.658,Z 462.032,A -85,B 0,C 180,E1 -6597.142,E2 -6597.142} C_VEL
LIN {X 0,Y 490.042,Z 448.55,A -85,B 0,C 180,E1 -6600.13,E2 -6600.13} C_VEL
LIN {X 0,Y 490.377,Z 434.322,A -85,B 0,C 180,E1 -6603.394,E2 -6603.394} C_VEL
LIN {X 0,Y 490.875,Z 423.595,A -85,B 0,C 180,E1 -6605.945,E2 -6605.945} C_VEL
LIN {X 0,Y 490.453,Z 419.45,A -85,B 0,C 180,E1 -6607.002,E2 -6607.002} C_VEL
LIN {X 0,Y 488.762,Z 410.606,A -85,B 0,C 180,E1 -6609.448,E2 -6609.448} C_VEL
LIN {X 0,Y 488.712,Z 410.611,A -85,B 0,C 180,E1 -6612.827,E2 -6612.827} C_VEL
LIN {X 0,Y 488.706,Z 410.612,A -85,B 0,C 180,E1 -6615.976,E2 -6615.976} C_VEL
LIN {X 0,Y 488.722,Z 410.611,A -85,B 0,C 180,E1 -6618.586,E2 -6618.586} C_VEL
LIN {X 0,Y 488.684,Z 410.615,A -85,B 0,C 180,E1 -6621.8,E2 -6621.8} C_VEL
LIN {X 0,Y 488.732,Z 410.607,A -85,B 0,C 180,E1 -6625.052,E2 -6625.052} C_VEL
LIN {X 0,Y 488.71,Z 410.612,A -85,B 0,C 180,E1 -6628.045,E2 -6628.045} C_VEL
LIN {X 0,Y 488.727,Z 410.607,A -85,B 0,C 180,E1 -6630.73,E2 -6630.73} C_VEL
LIN {X 0,Y 488.757,Z 410.605,A -85,B 0,C 180,E1 -6633.528,E2 -6633.528} C_VEL
LIN {X 0,Y 488.683,Z 410.615,A -85,B 0,C 180,E1 -6636.254,E2 -6636.254} C_VEL
LIN {X 0,Y 488.75,Z 410.606,A -85,B 0,C 180,E1 -6639.176,E2 -6639.176} C_VEL
LIN {X 0,Y 488.763,Z 410.605,A -85,B 0,C 180,E1 -6641.628,E2 -6641.628} C_VEL
LIN {X 0,Y 488.766,Z 410.602,A -85,B 0,C 180,E1 -6645,E2 -6645} C_VEL
LIN {X 0,Y 488.834,Z 410.595,A -85,B 0,C 180,E1 -6648.388,E2 -6648.388} C_VEL
LIN {X 0,Y 488.789,Z 410.603,A -85,B 0,C 180,E1 -6651.733,E2 -6651.733} C_VEL
LIN {X 0,Y 488.86,Z 410.592,A -85,B 0,C 180,E1 -6654.224,E2 -6654.224} C_VEL
LIN {X 0,Y 488.967,Z 410.579,A -85,B 0,C 180,E1 -6657.529,E2 -6657.529} C_VEL
LIN {X 0,Y 488.96,Z 410.578,A -85,B 0,C 180,E1 -6660.824,E2 -6660.824} C_VEL
LIN {X 0,Y 488.965,Z 410.577,A -85,B 0,C 180,E1 -6662.471,E2 -6662.471} C_VEL
LIN {X 0,Y 488.854,Z 410.593,A -85,B 0,C 180,E1 -6665.776,E2 -6665.776} C_VEL
LIN {X 0,Y 488.79,Z 410.6,A -85,B 0,C 180,E1 -6668.267,E2 -6668.267} C_VEL
LIN {X 0,Y 488.834,Z 410.597,A -85,B 0,C 180,E1 -6671.612,E2 -6671.612} C_VEL
LIN {X 0,Y 488.767,Z 410.604,A -85,B 0,C 180,E1 -6675,E2 -6675} C_VEL
LIN {X 0,Y 488.759,Z 410.603,A -85,B 0,C 180,E1 -6678.442,E2 -6678.442} C_VEL
LIN {X 0,Y 488.711,Z 410.611,A -85,B 0,C 180,E1 -6681.071,E2 -6681.071} C_VEL
LIN {X 0,Y 488.692,Z 410.613,A -85,B 0,C 180,E1 -6683.746,E2 -6683.746} C_VEL
LIN {X 0,Y 488.796,Z 410.601,A -85,B 0,C 180,E1 -6686.944,E2 -6686.944} C_VEL
LIN {X 0,Y 488.714,Z 410.608,A -85,B 0,C 180,E1 -6690.363,E2 -6690.363} C_VEL
LIN {X 0,Y 488.739,Z 410.608,A -85,B 0,C 180,E1 -6693.484,E2 -6693.484} C_VEL
LIN {X 0,Y 488.686,Z 410.613,A -85,B 0,C 180,E1 -6696.354,E2 -6696.354} C_VEL
LIN {X 0,Y 488.704,Z 410.614,A -85,B 0,C 180,E1 -6699.254,E2 -6699.254} C_VEL
LIN {X 0,Y 488.727,Z 410.608,A -85,B 0,C 180,E1 -6701.602,E2 -6701.602} C_VEL
LIN {X 0,Y 488.716,Z 410.612,A -85,B 0,C 180,E1 -6704.801,E2 -6704.801} C_VEL
LIN {X 0,Y 488.739,Z 410.608,A -85,B 0,C 180,E1 -6707.479,E2 -6707.479} C_VEL
LIN {X 0,Y 488.753,Z 410.606,A -85,B 0,C 180,E1 -6710.75,E2 -6710.75} C_VEL
LIN {X 0,Y 488.681,Z 410.613,A -85,B 0,C 180,E1 -6713.868,E2 -6713.868} C_VEL
LIN {X 0,Y 488.742,Z 410.608,A -85,B 0,C 180,E1 -6716.877,E2 -6716.877} C_VEL
LIN {X 0,Y 488.728,Z 410.607,A -85,B 0,C 180,E1 -6719.781,E2 -6719.781} C_VEL
LIN {X 0,Y 488.796,Z 410.601,A -85,B 0,C 180,E1 -6723.056,E2 -6723.056} C_VEL
LIN {X 0,Y 488.747,Z 410.605,A -85,B 0,C 180,E1 -6724.343,E2 -6724.343} C_VEL
LIN {X 0,Y 488.103,Z 410.689,A -85,B 0,C 180,E1 -6725.03,E2 -6725.03} C_VEL
LIN {X 0,Y 485.236,Z 411.047,A -85,B 0,C 180,E1 -6726.147,E2 -6726.147} C_VEL
LIN {X 0,Y 482.791,Z 411.349,A -85,B 0,C 180,E1 -6727.046,E2 -6727.046} C_VEL
LIN {X 0,Y 481.732,Z 411.479,A -85,B 0,C 180,E1 -6727.742,E2 -6727.742} C_VEL
LIN {X 0,Y 481.643,Z 411.489,A -85,B 0,C 180,E1 -6727.977,E2 -6727.977} C_VEL
LIN {X 0,Y 481.709,Z 411.484,A -85,B 0,C 180,E1 -6730.393,E2 -6730.393} C_VEL
LIN {X 0,Y 481.692,Z 411.487,A -85,B 0,C 180,E1 -6733.034,E2 -6733.034} C_VEL
LIN {X 0,Y 481.713,Z 411.55,A -85,B 0,C 180,E1 -6735.855,E2 -6735.855} C_VEL
LIN {X 0,Y 484.036,Z 419.781,A -85,B 0,C 180,E1 -6736.353,E2 -6736.353} C_VEL
LIN {X 0,Y 483.885,Z 430.578,A -85,B 0,C 180,E1 -6737.021,E2 -6737.021} C_VEL
LIN {X 0,Y 483.499,Z 441.078,A -85,B 0,C 180,E1 -6737.833,E2 -6737.833} C_VEL
LIN {X 0,Y 483.189,Z 449.922,A -85,B 0,C 180,E1 -6738.676,E2 -6738.676} C_VEL
LIN {X 0,Y 482.768,Z 458.992,A -85,B 0,C 180,E1 -6739.727,E2 -6739.727} C_VEL
LIN {X 0,Y 482.329,Z 467.772,A -85,B 0,C 180,E1 -6740.988,E2 -6740.988} C_VEL
LIN {X 0,Y 482.033,Z 474.821,A -85,B 0,C 180,E1 -6742.249,E2 -6742.249} C_VEL
LIN {X 0,Y 481.854,Z 479.569,A -85,B 0,C 180,E1 -6743.299,E2 -6743.299} C_VEL
LIN {X 0,Y 481.585,Z 484.19,A -85,B 0,C 180,E1 -6744.557,E2 -6744.557} C_VEL
LIN {X 0,Y 481.476,Z 487.712,A -85,B 0,C 180,E1 -6745.815,E2 -6745.815} C_VEL
LIN {X 0,Y 481.384,Z 489.537,A -85,B 0,C 180,E1 -6746.652,E2 -6746.652} C_VEL
LIN {X 0,Y 481.282,Z 490.918,A -85,B 0,C 180,E1 -6747.489,E2 -6747.489} C_VEL
LIN {X 0,Y 481.299,Z 491.885,A -85,B 0,C 180,E1 -6748.326,E2 -6748.326} C_VEL
LIN {X 0,Y 481.215,Z 492.725,A -85,B 0,C 180,E1 -6750,E2 -6750} C_VEL
LIN {X 0,Y 481.299,Z 491.967,A -85,B 0,C 180,E1 -6751.673,E2 -6751.673} C_VEL
LIN {X 0,Y 481.379,Z 489.703,A -85,B 0,C 180,E1 -6753.348,E2 -6753.348} C_VEL
LIN {X 0,Y 481.535,Z 486.898,A -85,B 0,C 180,E1 -6754.604,E2 -6754.604} C_VEL
LIN {X 0,Y 481.714,Z 483.096,A -85,B 0,C 180,E1 -6755.862,E2 -6755.862} C_VEL
LIN {X 0,Y 481.859,Z 477.198,A -85,B 0,C 180,E1 -6757.344,E2 -6757.344} C_VEL
LIN {X 0,Y 482.227,Z 470.802,A -85,B 0,C 180,E1 -6758.591,E2 -6758.591} C_VEL
LIN {X 0,Y 482.628,Z 462.784,A -85,B 0,C 180,E1 -6759.852,E2 -6759.852} C_VEL
LIN {X 0,Y 482.926,Z 454.575,A -85,B 0,C 180,E1 -6760.905,E2 -6760.905} C_VEL
LIN {X 0,Y 483.385,Z 444.395,A -85,B 0,C 180,E1 -6761.957,E2 -6761.957} C_VEL
LIN {X 0,Y 483.791,Z 433.916,A -85,B 0,C 180,E1 -6762.828,E2 -6762.828} C_VEL
LIN {X 0,Y 484.11,Z 423.238,A -85,B 0,C 180,E1 -6763.538,E2 -6763.538} C_VEL
LIN {X 0,Y 483.963,Z 419.5,A -85,B 0,C 180,E1 -6763.756,E2 -6763.756} C_VEL
LIN {X 0,Y 481.701,Z 411.477,A -85,B 0,C 180,E1 -6764.253,E2 -6764.253} C_VEL
LIN {X 0,Y 481.683,Z 411.487,A -85,B 0,C 180,E1 -6766.966,E2 -6766.966} C_VEL
LIN {X 0,Y 481.708,Z 411.484,A -85,B 0,C 180,E1 -6769.607,E2 -6769.607} C_VEL
LIN {X 0,Y 481.657,Z 411.488,A -85,B 0,C 180,E1 -6772.295,E2 -6772.295} C_VEL
LIN {X 0,Y 481.716,Z 411.484,A -85,B 0,C 180,E1 -6775.237,E2 -6775.237} C_VEL
LIN {X 0,Y 481.706,Z 411.482,A -85,B 0,C 180,E1 -6777.832,E2 -6777.832} C_VEL
LIN {X 0,Y 481.649,Z 411.491,A -85,B 0,C 180,E1 -6780.711,E2 -6780.711} C_VEL
LIN {X 0,Y 481.7,Z 411.484,A -85,B 0,C 180,E1 -6783.733,E2 -6783.733} C_VEL
LIN {X 0,Y 481.633,Z 411.492,A -85,B 0,C 180,E1 -6786.746,E2 -6786.746} C_VEL
LIN {X 0,Y 481.696,Z 411.483,A -85,B 0,C 180,E1 -6789.939,E2 -6789.939} C_VEL
LIN {X 0,Y 481.687,Z 411.487,A -85,B 0,C 180,E1 -6793.295,E2 -6793.295} C_VEL
LIN {X 0,Y 481.673,Z 411.488,A -85,B 0,C 180,E1 -6796.848,E2 -6796.848} C_VEL
LIN {X 0,Y 481.679,Z 411.485,A -85,B 0,C 180,E1 -6800.06,E2 -6800.06} C_VEL
LIN {X 0,Y 481.628,Z 411.493,A -85,B 0,C 180,E1 -6803.253,E2 -6803.253} C_VEL
LIN {X 0,Y 481.712,Z 411.483,A -85,B 0,C 180,E1 -6806.33,E2 -6806.33} C_VEL
LIN {X 0,Y 481.654,Z 411.488,A -85,B 0,C 180,E1 -6809.417,E2 -6809.417} C_VEL
LIN {X 0,Y 481.703,Z 411.482,A -85,B 0,C 180,E1 -6812.168,E2 -6812.168} C_VEL
LIN {X 0,Y 481.696,Z 411.485,A -85,B 0,C 180,E1 -6814.969,E2 -6814.969} C_VEL
LIN {X 0,Y 481.651,Z 411.489,A -85,B 0,C 180,E1 -6817.705,E2 -6817.705} C_VEL
LIN {X 0,Y 481.712,Z 411.483,A -85,B 0,C 180,E1 -6820.393,E2 -6820.393} C_VEL
LIN {X 0,Y 481.696,Z 411.485,A -85,B 0,C 180,E1 -6823.034,E2 -6823.034} C_VEL
LIN {X 0,Y 481.693,Z 411.483,A -85,B 0,C 180,E1 -6825.639,E2 -6825.639} C_VEL
LIN {X 0,Y 481.798,Z 411.472,A -85,B 0,C 180,E1 -6828.216,E2 -6828.216} C_VEL
LIN {X 0,Y 481.744,Z 411.478,A -85,B 0,C 180,E1 -6831.611,E2 -6831.611} C_VEL
LIN {X 0,Y 481.819,Z 411.469,A -85,B 0,C 180,E1 -6834.14,E2 -6834.14} C_VEL
LIN {X 0,Y 481.931,Z 411.453,A -85,B 0,C 180,E1 -6837.493,E2 -6837.493} C_VEL
LIN {X 0,Y 481.91,Z 411.459,A -85,B 0,C 180,E1 -6840.836,E2 -6840.836} C_VEL
LIN {X 0,Y 481.932,Z 411.456,A -85,B 0,C 180,E1 -6842.507,E2 -6842.507} C_VEL
LIN {X 0,Y 481.82,Z 411.469,A -85,B 0,C 180,E1 -6845.86,E2 -6845.86} C_VEL
LIN {X 0,Y 481.742,Z 411.481,A -85,B 0,C 180,E1 -6848.389,E2 -6848.389} C_VEL
LIN {X 0,Y 481.798,Z 411.472,A -85,B 0,C 180,E1 -6851.784,E2 -6851.784} C_VEL
LIN {X 0,Y 481.746,Z 411.476,A -85,B 0,C 180,E1 -6855.224,E2 -6855.224} C_VEL
LIN {X 0,Y 481.716,Z 411.483,A -85,B 0,C 180,E1 -6858.722,E2 -6858.722} C_VEL
LIN {X 0,Y 481.648,Z 411.49,A -85,B 0,C 180,E1 -6861.395,E2 -6861.395} C_VEL
LIN {X 0,Y 481.664,Z 411.49,A -85,B 0,C 180,E1 -6864.114,E2 -6864.114} C_VEL
LIN {X 0,Y 481.75,Z 411.476,A -85,B 0,C 180,E1 -6867.139,E2 -6867.139} C_VEL
LIN {X 0,Y 481.682,Z 411.488,A -85,B 0,C 180,E1 -6869.741,E2 -6869.741} C_VEL
LIN {X 0,Y 481.676,Z 411.487,A -85,B 0,C 180,E1 -6872.674,E2 -6872.674} C_VEL
LIN {X 0,Y 481.645,Z 411.491,A -85,B 0,C 180,E1 -6875.709,E2 -6875.709} C_VEL
LIN {X 0,Y 481.673,Z 411.486,A -85,B 0,C 180,E1 -6878.859,E2 -6878.859} C_VEL
LIN {X 0,Y 481.664,Z 411.489,A -85,B 0,C 180,E1 -6881.914,E2 -6881.914} C_VEL
LIN {X 0,Y 481.663,Z 411.492,A -85,B 0,C 180,E1 -6884.457,E2 -6884.457} C_VEL
LIN {X 0,Y 481.651,Z 411.49,A -85,B 0,C 180,E1 -6887.84,E2 -6887.84} C_VEL
LIN {X 0,Y 481.731,Z 411.535,A -85,B 0,C 180,E1 -6890.347,E2 -6890.347} C_VEL
LIN {X 0,Y 483.836,Z 422.9,A -85,B 0,C 180,E1 -6893.448,E2 -6893.448} C_VEL
LIN {X 0,Y 483.725,Z 429.074,A -85,B 0,C 180,E1 -6894.978,E2 -6894.978} C_VEL
LIN {X 0,Y 483.203,Z 443.596,A -85,B 0,C 180,E1 -6898.425,E2 -6898.425} C_VEL
LIN {X 0,Y 482.827,Z 457.181,A -85,B 0,C 180,E1 -6901.529,E2 -6901.529} C_VEL
LIN {X 0,Y 482.445,Z 470.888,A -85,B 0,C 180,E1 -6904.58,E2 -6904.58} C_VEL
LIN {X 0,Y 482.142,Z 484.202,A -85,B 0,C 180,E1 -6907.503,E2 -6907.503} C_VEL
LIN {X 0,Y 481.818,Z 499.482,A -85,B 0,C 180,E1 -6910.841,E2 -6910.841} C_VEL
LIN {X 0,Y 481.539,Z 513.485,A -85,B 0,C 180,E1 -6913.901,E2 -6913.901} C_VEL
LIN {X 0,Y 481.44,Z 518.554,A -85,B 0,C 180,E1 -6915.01,E2 -6915.01} C_VEL
LIN {X 0,Y 482.891,Z 533.833,A -85,B 0,C 180,E1 -6915.42,E2 -6915.42} C_VEL
LIN {X 0,Y 483.69,Z 539.887,A -85,B 0,C 180,E1 -6915.646,E2 -6915.646} C_VEL
LIN {X 0,Y 483.256,Z 552.02,A -85,B 0,C 180,E1 -6916.169,E2 -6916.169} C_VEL
LIN {X 0,Y 482.814,Z 564.347,A -85,B 0,C 180,E1 -6916.886,E2 -6916.886} C_VEL
LIN {X 0,Y 482.46,Z 575.17,A -85,B 0,C 180,E1 -6917.686,E2 -6917.686} C_VEL
LIN {X 0,Y 482.006,Z 585.698,A -85,B 0,C 180,E1 -6918.648,E2 -6918.648} C_VEL
LIN {X 0,Y 481.643,Z 595.043,A -85,B 0,C 180,E1 -6919.703,E2 -6919.703} C_VEL
LIN {X 0,Y 481.377,Z 604.178,A -85,B 0,C 180,E1 -6920.97,E2 -6920.97} C_VEL
LIN {X 0,Y 481.197,Z 611.551,A -85,B 0,C 180,E1 -6922.236,E2 -6922.236} C_VEL
LIN {X 0,Y 481.092,Z 618.168,A -85,B 0,C 180,E1 -6923.68,E2 -6923.68} C_VEL
LIN {X 0,Y 481.072,Z 622.751,A -85,B 0,C 180,E1 -6924.971,E2 -6924.971} C_VEL
LIN {X 0,Y 481.076,Z 625.117,A -85,B 0,C 180,E1 -6925.811,E2 -6925.811} C_VEL
LIN {X 0,Y 481.051,Z 627.033,A -85,B 0,C 180,E1 -6926.65,E2 -6926.65} C_VEL
LIN {X 0,Y 481.032,Z 628.471,A -85,B 0,C 180,E1 -6927.488,E2 -6927.488} C_VEL
LIN {X 0,Y 480.992,Z 629.492,A -85,B 0,C 180,E1 -6928.325,E2 -6928.325} C_VEL
LIN {X 0,Y 481.047,Z 630.35,A -85,B 0,C 180,E1 -6930,E2 -6930} C_VEL
LIN {X 0,Y 480.992,Z 629.494,A -85,B 0,C 180,E1 -6931.675,E2 -6931.675} C_VEL
LIN {X 0,Y 481.032,Z 628.474,A -85,B 0,C 180,E1 -6932.512,E2 -6932.512} C_VEL
LIN {X 0,Y 481.051,Z 627.036,A -85,B 0,C 180,E1 -6933.35,E2 -6933.35} C_VEL
LIN {X 0,Y 481.047,Z 624.011,A -85,B 0,C 180,E1 -6934.609,E2 -6934.609} C_VEL
LIN {X 0,Y 481.125,Z 619.93,A -85,B 0,C 180,E1 -6935.869,E2 -6935.869} C_VEL
LIN {X 0,Y 481.153,Z 613.642,A -85,B 0,C 180,E1 -6937.343,E2 -6937.343} C_VEL
LIN {X 0,Y 481.309,Z 606.801,A -85,B 0,C 180,E1 -6938.608,E2 -6938.608} C_VEL
LIN {X 0,Y 481.524,Z 598.33,A -85,B 0,C 180,E1 -6939.875,E2 -6939.875} C_VEL
LIN {X 0,Y 481.867,Z 589.676,A -85,B 0,C 180,E1 -6940.93,E2 -6940.93} C_VEL
LIN {X 0,Y 482.297,Z 579.314,A -85,B 0,C 180,E1 -6941.958,E2 -6941.958} C_VEL
LIN {X 0,Y 482.669,Z 568.484,A -85,B 0,C 180,E1 -6942.83,E2 -6942.83} C_VEL
LIN {X 0,Y 483.065,Z 556.971,A -85,B 0,C 180,E1 -6943.568,E2 -6943.568} C_VEL
LIN {X 0,Y 483.501,Z 545.192,A -85,B 0,C 180,E1 -6944.145,E2 -6944.145} C_VEL
LIN {X 0,Y 483.517,Z 538.307,A -85,B 0,C 180,E1 -6944.413,E2 -6944.413} C_VEL
LIN {X 0,Y 482.293,Z 527.397,A -85,B 0,C 180,E1 -6944.774,E2 -6944.774} C_VEL
LIN {X 0,Y 481.441,Z 518.523,A -85,B 0,C 180,E1 -6944.99,E2 -6944.99} C_VEL
LIN {X 0,Y 481.709,Z 504.005,A -85,B 0,C 180,E1 -6948.175,E2 -6948.175} C_VEL
LIN {X 0,Y 482.009,Z 489.322,A -85,B 0,C 180,E1 -6951.378,E2 -6951.378} C_VEL
LIN {X 0,Y 482.333,Z 475.937,A -85,B 0,C 180,E1 -6954.307,E2 -6954.307} C_VEL
LIN {X 0,Y 482.648,Z 462.197,A -85,B 0,C 180,E1 -6957.346,E2 -6957.346} C_VEL
LIN {X 0,Y 483.055,Z 448.809,A -85,B 0,C 180,E1 -6960.37,E2 -6960.37} C_VEL
LIN {X 0,Y 483.423,Z 435.246,A -85,B 0,C 180,E1 -6963.535,E2 -6963.535} C_VEL
LIN {X 0,Y 483.916,Z 423.905,A -85,B 0,C 180,E1 -6966.286,E2 -6966.286} C_VEL
LIN {X 0,Y 482.712,Z 416.855,A -85,B 0,C 180,E1 -6968.167,E2 -6968.167} C_VEL
LIN {X 0,Y 481.733,Z 411.482,A -85,B 0,C 180,E1 -6969.693,E2 -6969.693} C_VEL
LIN {X 0,Y 481.646,Z 411.491,A -85,B 0,C 180,E1 -6973.149,E2 -6973.149} C_VEL
LIN {X 0,Y 481.662,Z 411.489,A -85,B 0,C 180,E1 -6975.641,E2 -6975.641} C_VEL
LIN {X 0,Y 481.666,Z 411.49,A -85,B 0,C 180,E1 -6978.959,E2 -6978.959} C_VEL
LIN {X 0,Y 481.659,Z 411.491,A -85,B 0,C 180,E1 -6981.993,E2 -6981.993} C_VEL
LIN {X 0,Y 481.696,Z 411.484,A -85,B 0,C 180,E1 -6985.318,E2 -6985.318} C_VEL
LIN {X 0,Y 481.651,Z 411.491,A -85,B 0,C 180,E1 -6988.312,E2 -6988.312} C_VEL
LIN {X 0,Y 481.704,Z 411.482,A -85,B 0,C 180,E1 -6991.219,E2 -6991.219} C_VEL
LIN {X 0,Y 481.693,Z 411.486,A -85,B 0,C 180,E1 -6994.042,E2 -6994.042} C_VEL
LIN {X 0,Y 481.677,Z 411.486,A -85,B 0,C 180,E1 -6996.812,E2 -6996.812} C_VEL
LIN {X 0,Y 481.701,Z 411.484,A -85,B 0,C 180,E1 -6999.503,E2 -6999.503} C_VEL
LIN {X 0,Y 481.712,Z 411.483,A -85,B 0,C 180,E1 -7002.159,E2 -7002.159} C_VEL
LIN {X 0,Y 481.747,Z 411.476,A -85,B 0,C 180,E1 -7004.776,E2 -7004.776} C_VEL
LIN {X 0,Y 481.799,Z 411.473,A -85,B 0,C 180,E1 -7008.216,E2 -7008.216} C_VEL
LIN {X 0,Y 481.743,Z 411.48,A -85,B 0,C 180,E1 -7011.611,E2 -7011.611} C_VEL
LIN {X 0,Y 481.821,Z 411.469,A -85,B 0,C 180,E1 -7014.14,E2 -7014.14} C_VEL
LIN {X 0,Y 481.934,Z 411.456,A -85,B 0,C 180,E1 -7017.493,E2 -7017.493} C_VEL
LIN {X 0,Y 481.911,Z 411.456,A -85,B 0,C 180,E1 -7020.836,E2 -7020.836} C_VEL
LIN {X 0,Y 481.932,Z 411.453,A -85,B 0,C 180,E1 -7022.507,E2 -7022.507} C_VEL
LIN {X 0,Y 481.815,Z 411.47,A -85,B 0,C 180,E1 -7025.86,E2 -7025.86} C_VEL
LIN {X 0,Y 481.745,Z 411.477,A -85,B 0,C 180,E1 -7028.389,E2 -7028.389} C_VEL
LIN {X 0,Y 481.8,Z 411.472,A -85,B 0,C 180,E1 -7031.784,E2 -7031.784} C_VEL
LIN {X 0,Y 481.747,Z 411.479,A -85,B 0,C 180,E1 -7035.224,E2 -7035.224} C_VEL
LIN {X 0,Y 481.717,Z 411.481,A -85,B 0,C 180,E1 -7038.722,E2 -7038.722} C_VEL
LIN {X 0,Y 481.65,Z 411.492,A -85,B 0,C 180,E1 -7041.395,E2 -7041.395} C_VEL
LIN {X 0,Y 481.678,Z 411.486,A -85,B 0,C 180,E1 -7044.113,E2 -7044.113} C_VEL
LIN {X 0,Y 481.751,Z 411.478,A -85,B 0,C 180,E1 -7047.139,E2 -7047.139} C_VEL
LIN {X 0,Y 481.683,Z 411.486,A -85,B 0,C 180,E1 -7049.741,E2 -7049.741} C_VEL
LIN {X 0,Y 481.677,Z 411.486,A -85,B 0,C 180,E1 -7052.674,E2 -7052.674} C_VEL
LIN {X 0,Y 481.64,Z 411.492,A -85,B 0,C 180,E1 -7055.709,E2 -7055.709} C_VEL
LIN {X 0,Y 481.674,Z 411.488,A -85,B 0,C 180,E1 -7058.859,E2 -7058.859} C_VEL
LIN {X 0,Y 481.666,Z 411.487,A -85,B 0,C 180,E1 -7061.914,E2 -7061.914} C_VEL
LIN {X 0,Y 481.664,Z 411.487,A -85,B 0,C 180,E1 -7064.457,E2 -7064.457} C_VEL
LIN {X 0,Y 481.693,Z 411.487,A -85,B 0,C 180,E1 -7066.846,E2 -7066.846} C_VEL
LIN {X 0,Y 481.697,Z 411.483,A -85,B 0,C 180,E1 -7070.061,E2 -7070.061} C_VEL
LIN {X 0,Y 481.639,Z 411.491,A -85,B 0,C 180,E1 -7072.203,E2 -7072.203} C_VEL
LIN {X 0,Y 481.692,Z 411.485,A -85,B 0,C 180,E1 -7075.318,E2 -7075.318} C_VEL
LIN {X 0,Y 481.648,Z 411.49,A -85,B 0,C 180,E1 -7078.312,E2 -7078.312} C_VEL
LIN {X 0,Y 481.704,Z 411.485,A -85,B 0,C 180,E1 -7081.219,E2 -7081.219} C_VEL
LIN {X 0,Y 481.705,Z 411.483,A -85,B 0,C 180,E1 -7084.043,E2 -7084.043} C_VEL
LIN {X 0,Y 481.678,Z 411.489,A -85,B 0,C 180,E1 -7086.812,E2 -7086.812} C_VEL
LIN {X 0,Y 481.643,Z 411.489,A -85,B 0,C 180,E1 -7087.977,E2 -7087.977} C_VEL
LIN {X 0,Y 480.974,Z 411.576,A -85,B 0,C 180,E1 -7088.675,E2 -7088.675} C_VEL
LIN {X 0,Y 478.146,Z 411.925,A -85,B 0,C 180,E1 -7089.81,E2 -7089.81} C_VEL
LIN {X 0,Y 475.762,Z 412.225,A -85,B 0,C 180,E1 -7090.724,E2 -7090.724} C_VEL
LIN {X 0,Y 474.74,Z 412.35,A -85,B 0,C 180,E1 -7091.43,E2 -7091.43} C_VEL
LIN {X 0,Y 474.658,Z 412.36,A -85,B 0,C 180,E1 -7091.669,E2 -7091.669} C_VEL
LIN {X 0,Y 474.704,Z 412.356,A -85,B 0,C 180,E1 -7094.544,E2 -7094.544} C_VEL
LIN {X 0,Y 474.674,Z 412.36,A -85,B 0,C 180,E1 -7095.613,E2 -7095.613} C_VEL
LIN {X 0,Y 477.06,Z 420.817,A -85,B 0,C 180,E1 -7096.149,E2 -7096.149} C_VEL
LIN {X 0,Y 477.219,Z 425.078,A -85,B 0,C 180,E1 -7096.406,E2 -7096.406} C_VEL
LIN {X 0,Y 476.81,Z 436.933,A -85,B 0,C 180,E1 -7097.227,E2 -7097.227} C_VEL
LIN {X 0,Y 476.39,Z 447.792,A -85,B 0,C 180,E1 -7098.188,E2 -7098.188} C_VEL
LIN {X 0,Y 475.933,Z 458.323,A -85,B 0,C 180,E1 -7099.363,E2 -7099.363} C_VEL
LIN {X 0,Y 475.579,Z 466.076,A -85,B 0,C 180,E1 -7100.43,E2 -7100.43} C_VEL
LIN {X 0,Y 475.165,Z 473.656,A -85,B 0,C 180,E1 -7101.708,E2 -7101.708} C_VEL
LIN {X 0,Y 474.879,Z 480.575,A -85,B 0,C 180,E1 -7103.2,E2 -7103.2} C_VEL
LIN {X 0,Y 474.598,Z 485.196,A -85,B 0,C 180,E1 -7104.476,E2 -7104.476} C_VEL
LIN {X 0,Y 474.467,Z 488.719,A -85,B 0,C 180,E1 -7105.753,E2 -7105.753} C_VEL
LIN {X 0,Y 474.368,Z 490.543,A -85,B 0,C 180,E1 -7106.602,E2 -7106.602} C_VEL
LIN {X 0,Y 474.261,Z 491.924,A -85,B 0,C 180,E1 -7107.452,E2 -7107.452} C_VEL
LIN {X 0,Y 474.281,Z 492.889,A -85,B 0,C 180,E1 -7108.302,E2 -7108.302} C_VEL
LIN {X 0,Y 474.19,Z 493.73,A -85,B 0,C 180,E1 -7110,E2 -7110} C_VEL
LIN {X 0,Y 474.281,Z 492.97,A -85,B 0,C 180,E1 -7111.698,E2 -7111.698} C_VEL
LIN {X 0,Y 474.362,Z 490.707,A -85,B 0,C 180,E1 -7113.397,E2 -7113.397} C_VEL
LIN {X 0,Y 474.529,Z 487.902,A -85,B 0,C 180,E1 -7114.672,E2 -7114.672} C_VEL
LIN {X 0,Y 474.746,Z 484.096,A -85,B 0,C 180,E1 -7115.948,E2 -7115.948} C_VEL
LIN {X 0,Y 474.888,Z 478.204,A -85,B 0,C 180,E1 -7117.451,E2 -7117.451} C_VEL
LIN {X 0,Y 475.281,Z 471.804,A -85,B 0,C 180,E1 -7118.718,E2 -7118.718} C_VEL
LIN {X 0,Y 475.709,Z 463.786,A -85,B 0,C 180,E1 -7119.997,E2 -7119.997} C_VEL
LIN {X 0,Y 476.03,Z 455.576,A -85,B 0,C 180,E1 -7121.065,E2 -7121.065} C_VEL
LIN {X 0,Y 476.511,Z 445.395,A -85,B 0,C 180,E1 -7122.132,E2 -7122.132} C_VEL
LIN {X 0,Y 476.943,Z 434.902,A -85,B 0,C 180,E1 -7123.017,E2 -7123.017} C_VEL
LIN {X 0,Y 477.287,Z 424.234,A -85,B 0,C 180,E1 -7123.735,E2 -7123.735} C_VEL
LIN {X 0,Y 476.971,Z 420.521,A -85,B 0,C 180,E1 -7123.962,E2 -7123.962} C_VEL
LIN {X 0,Y 474.671,Z 412.352,A -85,B 0,C 180,E1 -7124.469,E2 -7124.469} C_VEL
LIN {X 0,Y 474.642,Z 412.364,A -85,B 0,C 180,E1 -7127.226,E2 -7127.226} C_VEL
LIN {X 0,Y 474.658,Z 412.363,A -85,B 0,C 180,E1 -7129.91,E2 -7129.91} C_VEL
LIN {X 0,Y 474.639,Z 412.365,A -85,B 0,C 180,E1 -7133.359,E2 -7133.359} C_VEL
LIN {X 0,Y 474.67,Z 412.358,A -85,B 0,C 180,E1 -7136.371,E2 -7136.371} C_VEL
LIN {X 0,Y 474.625,Z 412.366,A -85,B 0,C 180,E1 -7139.252,E2 -7139.252} C_VEL
LIN {X 0,Y 474.618,Z 412.364,A -85,B 0,C 180,E1 -7142.43,E2 -7142.43} C_VEL
LIN {X 0,Y 474.623,Z 412.366,A -85,B 0,C 180,E1 -7145.47,E2 -7145.47} C_VEL
LIN {X 0,Y 474.629,Z 412.365,A -85,B 0,C 180,E1 -7148.456,E2 -7148.456} C_VEL
LIN {X 0,Y 474.648,Z 412.363,A -85,B 0,C 180,E1 -7150.962,E2 -7150.962} C_VEL
LIN {X 0,Y 474.621,Z 412.364,A -85,B 0,C 180,E1 -7154.104,E2 -7154.104} C_VEL
LIN {X 0,Y 474.638,Z 412.364,A -85,B 0,C 180,E1 -7157.068,E2 -7157.068} C_VEL
LIN {X 0,Y 474.647,Z 412.362,A -85,B 0,C 180,E1 -7160.454,E2 -7160.454} C_VEL
LIN {X 0,Y 474.591,Z 412.368,A -85,B 0,C 180,E1 -7163.676,E2 -7163.676} C_VEL
LIN {X 0,Y 474.646,Z 412.364,A -85,B 0,C 180,E1 -7166.78,E2 -7166.78} C_VEL
LIN {X 0,Y 474.608,Z 412.365,A -85,B 0,C 180,E1 -7169.77,E2 -7169.77} C_VEL
LIN {X 0,Y 474.7,Z 412.357,A -85,B 0,C 180,E1 -7172.68,E2 -7172.68} C_VEL
LIN {X 0,Y 474.643,Z 412.362,A -85,B 0,C 180,E1 -7175.506,E2 -7175.506} C_VEL
LIN {X 0,Y 474.674,Z 412.359,A -85,B 0,C 180,E1 -7179.185,E2 -7179.185} C_VEL
LIN {X 0,Y 474.661,Z 412.359,A -85,B 0,C 180,E1 -7181.884,E2 -7181.884} C_VEL
LIN {X 0,Y 474.703,Z 412.356,A -85,B 0,C 180,E1 -7184.544,E2 -7184.544} C_VEL
LIN {X 0,Y 474.743,Z 412.35,A -85,B 0,C 180,E1 -7188.038,E2 -7188.038} C_VEL
LIN {X 0,Y 474.715,Z 412.353,A -85,B 0,C 180,E1 -7191.486,E2 -7191.486} C_VEL
LIN {X 0,Y 474.782,Z 412.346,A -85,B 0,C 180,E1 -7194.052,E2 -7194.052} C_VEL
LIN {X 0,Y 474.898,Z 412.329,A -85,B 0,C 180,E1 -7197.455,E2 -7197.455} C_VEL
LIN {X 0,Y 474.916,Z 412.329,A -85,B 0,C 180,E1 -7200,E2 -7200} C_VEL
LIN {X 0,Y 474.899,Z 412.332,A -85,B 0,C 180,E1 -7202.545,E2 -7202.545} C_VEL
LIN {X 0,Y 474.782,Z 412.346,A -85,B 0,C 180,E1 -7205.948,E2 -7205.948} C_VEL
LIN {X 0,Y 474.714,Z 412.355,A -85,B 0,C 180,E1 -7208.514,E2 -7208.514} C_VEL
LIN {X 0,Y 474.742,Z 412.352,A -85,B 0,C 180,E1 -7211.961,E2 -7211.961} C_VEL
LIN {X 0,Y 474.684,Z 412.358,A -85,B 0,C 180,E1 -7215.768,E2 -7215.768} C_VEL
LIN {X 0,Y 474.669,Z 412.359,A -85,B 0,C 180,E1 -7219.01,E2 -7219.01} C_VEL
LIN {X 0,Y 474.591,Z 412.37,A -85,B 0,C 180,E1 -7221.729,E2 -7221.729} C_VEL
LIN {X 0,Y 474.643,Z 412.363,A -85,B 0,C 180,E1 -7224.494,E2 -7224.494} C_VEL
LIN {X 0,Y 474.702,Z 412.354,A -85,B 0,C 180,E1 -7227.339,E2 -7227.339} C_VEL
LIN {X 0,Y 474.608,Z 412.366,A -85,B 0,C 180,E1 -7230.81,E2 -7230.81} C_VEL
LIN {X 0,Y 474.641,Z 412.365,A -85,B 0,C 180,E1 -7233.984,E2 -7233.984} C_VEL
LIN {X 0,Y 474.577,Z 412.37,A -85,B 0,C 180,E1 -7236.9,E2 -7236.9} C_VEL
LIN {X 0,Y 474.63,Z 412.365,A -85,B 0,C 180,E1 -7239.648,E2 -7239.648} C_VEL
LIN {X 0,Y 474.638,Z 412.366,A -85,B 0,C 180,E1 -7242.932,E2 -7242.932} C_VEL
LIN {X 0,Y 474.611,Z 412.367,A -85,B 0,C 180,E1 -7245.895,E2 -7245.895} C_VEL
LIN {X 0,Y 474.644,Z 412.361,A -85,B 0,C 180,E1 -7249.039,E2 -7249.039} C_VEL
LIN {X 0,Y 474.688,Z 412.451,A -85,B 0,C 180,E1 -7250.082,E2 -7250.082} C_VEL
LIN {X 0,Y 476.768,Z 423.197,A -85,B 0,C 180,E1 -7253.08,E2 -7253.08} C_VEL
LIN {X 0,Y 476.941,Z 427.306,A -85,B 0,C 180,E1 -7254.141,E2 -7254.141} C_VEL
LIN {X 0,Y 476.301,Z 441.421,A -85,B 0,C 180,E1 -7257.579,E2 -7257.579} C_VEL
LIN {X 0,Y 475.901,Z 454.358,A -85,B 0,C 180,E1 -7260.61,E2 -7260.61} C_VEL
LIN {X 0,Y 475.507,Z 467.821,A -85,B 0,C 180,E1 -7263.679,E2 -7263.679} C_VEL
LIN {X 0,Y 475.136,Z 482.355,A -85,B 0,C 180,E1 -7266.935,E2 -7266.935} C_VEL
LIN {X 0,Y 474.774,Z 497.568,A -85,B 0,C 180,E1 -7270.32,E2 -7270.32} C_VEL
LIN {X 0,Y 474.454,Z 510.561,A -85,B 0,C 180,E1 -7273.211,E2 -7273.211} C_VEL
LIN {X 0,Y 474.369,Z 517.575,A -85,B 0,C 180,E1 -7274.781,E2 -7274.781} C_VEL
LIN {X 0,Y 475.801,Z 533.248,A -85,B 0,C 180,E1 -7275.211,E2 -7275.211} C_VEL
LIN {X 0,Y 476.65,Z 541.561,A -85,B 0,C 180,E1 -7275.538,E2 -7275.538} C_VEL
LIN {X 0,Y 476.213,Z 554.008,A -85,B 0,C 180,E1 -7276.124,E2 -7276.124} C_VEL
LIN {X 0,Y 475.719,Z 566.006,A -85,B 0,C 180,E1 -7276.871,E2 -7276.871} C_VEL
LIN {X 0,Y 475.36,Z 576.499,A -85,B 0,C 180,E1 -7277.702,E2 -7277.702} C_VEL
LIN {X 0,Y 474.875,Z 586.661,A -85,B 0,C 180,E1 -7278.691,E2 -7278.691} C_VEL
LIN {X 0,Y 474.527,Z 595.681,A -85,B 0,C 180,E1 -7279.763,E2 -7279.763} C_VEL
LIN {X 0,Y 474.265,Z 604.511,A -85,B 0,C 180,E1 -7281.049,E2 -7281.049} C_VEL
LIN {X 0,Y 474.098,Z 611.584,A -85,B 0,C 180,E1 -7282.333,E2 -7282.333} C_VEL
LIN {X 0,Y 474.026,Z 617.496,A -85,B 0,C 180,E1 -7283.674,E2 -7283.674} C_VEL
LIN {X 0,Y 474.008,Z 621.736,A -85,B 0,C 180,E1 -7284.896,E2 -7284.896} C_VEL
LIN {X 0,Y 474.016,Z 624.104,A -85,B 0,C 180,E1 -7285.749,E2 -7285.749} C_VEL
LIN {X 0,Y 474.005,Z 626.023,A -85,B 0,C 180,E1 -7286.6,E2 -7286.6} C_VEL
LIN {X 0,Y 473.991,Z 627.463,A -85,B 0,C 180,E1 -7287.451,E2 -7287.451} C_VEL
LIN {X 0,Y 473.958,Z 628.486,A -85,B 0,C 180,E1 -7288.301,E2 -7288.301} C_VEL
LIN {X 0,Y 474.034,Z 629.347,A -85,B 0,C 180,E1 -7290,E2 -7290} C_VEL
LIN {X 0,Y 473.958,Z 628.487,A -85,B 0,C 180,E1 -7291.7,E2 -7291.7} C_VEL
LIN {X 0,Y 473.991,Z 627.466,A -85,B 0,C 180,E1 -7292.55,E2 -7292.55} C_VEL
LIN {X 0,Y 474.005,Z 626.027,A -85,B 0,C 180,E1 -7293.4,E2 -7293.4} C_VEL
LIN {X 0,Y 474.001,Z 623,A -85,B 0,C 180,E1 -7294.678,E2 -7294.678} C_VEL
LIN {X 0,Y 474.061,Z 618.914,A -85,B 0,C 180,E1 -7295.957,E2 -7295.957} C_VEL
LIN {X 0,Y 474.096,Z 612.625,A -85,B 0,C 180,E1 -7297.453,E2 -7297.453} C_VEL
LIN {X 0,Y 474.237,Z 605.778,A -85,B 0,C 180,E1 -7298.737,E2 -7298.737} C_VEL
LIN {X 0,Y 474.476,Z 597.306,A -85,B 0,C 180,E1 -7300.023,E2 -7300.023} C_VEL
LIN {X 0,Y 474.829,Z 588.65,A -85,B 0,C 180,E1 -7301.094,E2 -7301.094} C_VEL
LIN {X 0,Y 475.291,Z 578.573,A -85,B 0,C 180,E1 -7302.111,E2 -7302.111} C_VEL
LIN {X 0,Y 475.623,Z 568.904,A -85,B 0,C 180,E1 -7302.914,E2 -7302.914} C_VEL
LIN {X 0,Y 476.035,Z 557.734,A -85,B 0,C 180,E1 -7303.664,E2 -7303.664} C_VEL
LIN {X 0,Y 476.528,Z 545.397,A -85,B 0,C 180,E1 -7304.302,E2 -7304.302} C_VEL
LIN {X 0,Y 476.704,Z 540.239,A -85,B 0,C 180,E1 -7304.515,E2 -7304.515} C_VEL
LIN {X 0,Y 475.488,Z 529.493,A -85,B 0,C 180,E1 -7304.909,E2 -7304.909} C_VEL
LIN {X 0,Y 474.369,Z 517.558,A -85,B 0,C 180,E1 -7305.219,E2 -7305.219} C_VEL
LIN {X 0,Y 474.684,Z 502.265,A -85,B 0,C 180,E1 -7308.637,E2 -7308.637} C_VEL
LIN {X 0,Y 475.024,Z 486.387,A -85,B 0,C 180,E1 -7312.165,E2 -7312.165} C_VEL
LIN {X 0,Y 475.413,Z 471.959,A -85,B 0,C 180,E1 -7315.386,E2 -7315.386} C_VEL
LIN {X 0,Y 475.83,Z 457.402,A -85,B 0,C 180,E1 -7318.687,E2 -7318.687} C_VEL
LIN {X 0,Y 476.19,Z 444.881,A -85,B 0,C 180,E1 -7321.597,E2 -7321.597} C_VEL
LIN {X 0,Y 476.67,Z 432.12,A -85,B 0,C 180,E1 -7324.665,E2 -7324.665} C_VEL
LIN {X 0,Y 476.998,Z 425.248,A -85,B 0,C 180,E1 -7326.373,E2 -7326.373} C_VEL
LIN {X 0,Y 475.668,Z 417.572,A -85,B 0,C 180,E1 -7328.457,E2 -7328.457} C_VEL
LIN {X 0,Y 474.695,Z 412.356,A -85,B 0,C 180,E1 -7329.986,E2 -7329.986} C_VEL
LIN {X 0,Y 474.604,Z 412.366,A -85,B 0,C 180,E1 -7333.481,E2 -7333.481} C_VEL
LIN {X 0,Y 474.625,Z 412.367,A -85,B 0,C 180,E1 -7336.516,E2 -7336.516} C_VEL
LIN {X 0,Y 474.623,Z 412.364,A -85,B 0,C 180,E1 -7339.343,E2 -7339.343} C_VEL
LIN {X 0,Y 474.614,Z 412.366,A -85,B 0,C 180,E1 -7341.704,E2 -7341.704} C_VEL
LIN {X 0,Y 474.633,Z 412.364,A -85,B 0,C 180,E1 -7344.726,E2 -7344.726} C_VEL
LIN {X 0,Y 474.641,Z 412.364,A -85,B 0,C 180,E1 -7347.788,E2 -7347.788} C_VEL
LIN {X 0,Y 474.628,Z 412.363,A -85,B 0,C 180,E1 -7350.885,E2 -7350.885} C_VEL
LIN {X 0,Y 474.658,Z 412.362,A -85,B 0,C 180,E1 -7353.628,E2 -7353.628} C_VEL
LIN {X 0,Y 474.638,Z 412.363,A -85,B 0,C 180,E1 -7356.642,E2 -7356.642} C_VEL
LIN {X 0,Y 474.661,Z 412.362,A -85,B 0,C 180,E1 -7360.09,E2 -7360.09} C_VEL
LIN {X 0,Y 474.656,Z 412.36,A -85,B 0,C 180,E1 -7362.775,E2 -7362.775} C_VEL
LIN {X 0,Y 474.653,Z 412.363,A -85,B 0,C 180,E1 -7365.421,E2 -7365.421} C_VEL
LIN {X 0,Y 474.743,Z 412.351,A -85,B 0,C 180,E1 -7368.039,E2 -7368.039} C_VEL
LIN {X 0,Y 474.715,Z 412.355,A -85,B 0,C 180,E1 -7371.486,E2 -7371.486} C_VEL
LIN {X 0,Y 474.783,Z 412.346,A -85,B 0,C 180,E1 -7374.052,E2 -7374.052} C_VEL
LIN {X 0,Y 474.9,Z 412.332,A -85,B 0,C 180,E1 -7377.455,E2 -7377.455} C_VEL
LIN {X 0,Y 474.916,Z 412.33,A -85,B 0,C 180,E1 -7380,E2 -7380} C_VEL
LIN {X 0,Y 474.898,Z 412.329,A -85,B 0,C 180,E1 -7382.545,E2 -7382.545} C_VEL
LIN {X 0,Y 474.777,Z 412.347,A -85,B 0,C 180,E1 -7385.948,E2 -7385.948} C_VEL
LIN {X 0,Y 474.717,Z 412.353,A -85,B 0,C 180,E1 -7388.514,E2 -7388.514} C_VEL
LIN {X 0,Y 474.744,Z 412.35,A -85,B 0,C 180,E1 -7391.962,E2 -7391.962} C_VEL
LIN {X 0,Y 474.685,Z 412.359,A -85,B 0,C 180,E1 -7395.768,E2 -7395.768} C_VEL
LIN {X 0,Y 474.67,Z 412.36,A -85,B 0,C 180,E1 -7399.01,E2 -7399.01} C_VEL
LIN {X 0,Y 474.593,Z 412.369,A -85,B 0,C 180,E1 -7401.729,E2 -7401.729} C_VEL
LIN {X 0,Y 474.661,Z 412.36,A -85,B 0,C 180,E1 -7404.493,E2 -7404.493} C_VEL
LIN {X 0,Y 474.703,Z 412.357,A -85,B 0,C 180,E1 -7407.339,E2 -7407.339} C_VEL
LIN {X 0,Y 474.609,Z 412.367,A -85,B 0,C 180,E1 -7410.81,E2 -7410.81} C_VEL
LIN {X 0,Y 474.641,Z 412.362,A -85,B 0,C 180,E1 -7413.984,E2 -7413.984} C_VEL
LIN {X 0,Y 474.575,Z 412.372,A -85,B 0,C 180,E1 -7416.899,E2 -7416.899} C_VEL
LIN {X 0,Y 474.621,Z 412.365,A -85,B 0,C 180,E1 -7419.646,E2 -7419.646} C_VEL
LIN {X 0,Y 474.639,Z 412.364,A -85,B 0,C 180,E1 -7422.932,E2 -7422.932} C_VEL
LIN {X 0,Y 474.622,Z 412.364,A -85,B 0,C 180,E1 -7425.896,E2 -7425.896} C_VEL
LIN {X 0,Y 474.649,Z 412.364,A -85,B 0,C 180,E1 -7429.038,E2 -7429.038} C_VEL
LIN {X 0,Y 474.623,Z 412.365,A -85,B 0,C 180,E1 -7431.703,E2 -7431.703} C_VEL
LIN {X 0,Y 474.628,Z 412.365,A -85,B 0,C 180,E1 -7434.726,E2 -7434.726} C_VEL
LIN {X 0,Y 474.639,Z 412.361,A -85,B 0,C 180,E1 -7437.788,E2 -7437.788} C_VEL
LIN {X 0,Y 474.628,Z 412.366,A -85,B 0,C 180,E1 -7440.884,E2 -7440.884} C_VEL
LIN {X 0,Y 474.665,Z 412.359,A -85,B 0,C 180,E1 -7443.628,E2 -7443.628} C_VEL
LIN {X 0,Y 474.64,Z 412.364,A -85,B 0,C 180,E1 -7446.641,E2 -7446.641} C_VEL
LIN {X 0,Y 474.658,Z 412.36,A -85,B 0,C 180,E1 -7450.09,E2 -7450.09} C_VEL
LIN {X 0,Y 474.658,Z 412.36,A -85,B 0,C 180,E1 -7451.669,E2 -7451.669} C_VEL
LIN {X 0,Y 473.975,Z 412.448,A -85,B 0,C 180,E1 -7452.142,E2 -7452.142} C_VEL
LIN {X 0,Y 471.118,Z 412.803,A -85,B 0,C 180,E1 -7452.881,E2 -7452.881} C_VEL
LIN {X 0,Y 468.283,Z 413.155,A -85,B 0,C 180,E1 -7453.63,E2 -7453.63} C_VEL
LIN {X 0,Y 467.653,Z 413.233,A -85,B 0,C 180,E1 -7454.113,E2 -7454.113} C_VEL
LIN {X 0,Y 467.641,Z 413.33,A -85,B 0,C 180,E1 -7455.406,E2 -7455.406} C_VEL
LIN {X 0,Y 470.46,Z 423.751,A -85,B 0,C 180,E1 -7456.061,E2 -7456.061} C_VEL
LIN {X 0,Y 470.159,Z 434.327,A -85,B 0,C 180,E1 -7456.76,E2 -7456.76} C_VEL
LIN {X 0,Y 469.679,Z 445.432,A -85,B 0,C 180,E1 -7457.688,E2 -7457.688} C_VEL
LIN {X 0,Y 469.242,Z 455.79,A -85,B 0,C 180,E1 -7458.772,E2 -7458.772} C_VEL
LIN {X 0,Y 468.817,Z 464.174,A -85,B 0,C 180,E1 -7459.855,E2 -7459.855} C_VEL
LIN {X 0,Y 468.344,Z 472.304,A -85,B 0,C 180,E1 -7461.152,E2 -7461.152} C_VEL
LIN {X 0,Y 468.003,Z 478.442,A -85,B 0,C 180,E1 -7462.362,E2 -7462.362} C_VEL
LIN {X 0,Y 467.789,Z 484.799,A -85,B 0,C 180,E1 -7463.963,E2 -7463.963} C_VEL
LIN {X 0,Y 467.533,Z 488.683,A -85,B 0,C 180,E1 -7465.257,E2 -7465.257} C_VEL
LIN {X 0,Y 467.352,Z 491.549,A -85,B 0,C 180,E1 -7466.551,E2 -7466.551} C_VEL
LIN {X 0,Y 467.24,Z 492.929,A -85,B 0,C 180,E1 -7467.414,E2 -7467.414} C_VEL
LIN {X 0,Y 467.263,Z 493.894,A -85,B 0,C 180,E1 -7468.276,E2 -7468.276} C_VEL
LIN {X 0,Y 467.165,Z 494.734,A -85,B 0,C 180,E1 -7470,E2 -7470} C_VEL
LIN {X 0,Y 467.263,Z 493.974,A -85,B 0,C 180,E1 -7471.724,E2 -7471.724} C_VEL
LIN {X 0,Y 467.346,Z 491.712,A -85,B 0,C 180,E1 -7473.449,E2 -7473.449} C_VEL
LIN {X 0,Y 467.524,Z 488.906,A -85,B 0,C 180,E1 -7474.742,E2 -7474.742} C_VEL
LIN {X 0,Y 467.774,Z 485.097,A -85,B 0,C 180,E1 -7476.037,E2 -7476.037} C_VEL
LIN {X 0,Y 467.92,Z 479.209,A -85,B 0,C 180,E1 -7477.562,E2 -7477.562} C_VEL
LIN {X 0,Y 468.337,Z 472.806,A -85,B 0,C 180,E1 -7478.848,E2 -7478.848} C_VEL
LIN {X 0,Y 468.792,Z 464.787,A -85,B 0,C 180,E1 -7480.146,E2 -7480.146} C_VEL
LIN {X 0,Y 469.16,Z 456.573,A -85,B 0,C 180,E1 -7481.229,E2 -7481.229} C_VEL
LIN {X 0,Y 469.642,Z 446.395,A -85,B 0,C 180,E1 -7482.313,E2 -7482.313} C_VEL
LIN {X 0,Y 470.098,Z 435.896,A -85,B 0,C 180,E1 -7483.21,E2 -7483.21} C_VEL
LIN {X 0,Y 470.448,Z 425.234,A -85,B 0,C 180,E1 -7483.939,E2 -7483.939} C_VEL
LIN {X 0,Y 470.44,Z 423.431,A -85,B 0,C 180,E1 -7484.05,E2 -7484.05} C_VEL
LIN {X 0,Y 467.616,Z 413.232,A -85,B 0,C 180,E1 -7484.692,E2 -7484.692} C_VEL
LIN {X 0,Y 467.602,Z 413.241,A -85,B 0,C 180,E1 -7487.494,E2 -7487.494} C_VEL
LIN {X 0,Y 467.626,Z 413.239,A -85,B 0,C 180,E1 -7490.223,E2 -7490.223} C_VEL
LIN {X 0,Y 467.577,Z 413.243,A -85,B 0,C 180,E1 -7493.943,E2 -7493.943} C_VEL
LIN {X 0,Y 467.631,Z 413.237,A -85,B 0,C 180,E1 -7496.799,E2 -7496.799} C_VEL
LIN {X 0,Y 467.557,Z 413.245,A -85,B 0,C 180,E1 -7499.738,E2 -7499.738} C_VEL
LIN {X 0,Y 467.586,Z 413.242,A -85,B 0,C 180,E1 -7502.758,E2 -7502.758} C_VEL
LIN {X 0,Y 467.56,Z 413.244,A -85,B 0,C 180,E1 -7505.889,E2 -7505.889} C_VEL
LIN {X 0,Y 467.622,Z 413.24,A -85,B 0,C 180,E1 -7509.141,E2 -7509.141} C_VEL
LIN {X 0,Y 467.622,Z 413.238,A -85,B 0,C 180,E1 -7512.571,E2 -7512.571} C_VEL
LIN {X 0,Y 467.57,Z 413.242,A -85,B 0,C 180,E1 -7516.177,E2 -7516.177} C_VEL
LIN {X 0,Y 467.584,Z 413.244,A -85,B 0,C 180,E1 -7518.723,E2 -7518.723} C_VEL
LIN {X 0,Y 467.567,Z 413.243,A -85,B 0,C 180,E1 -7521.955,E2 -7521.955} C_VEL
LIN {X 0,Y 467.567,Z 413.245,A -85,B 0,C 180,E1 -7525.167,E2 -7525.167} C_VEL
LIN {X 0,Y 467.586,Z 413.241,A -85,B 0,C 180,E1 -7528.26,E2 -7528.26} C_VEL
LIN {X 0,Y 467.58,Z 413.243,A -85,B 0,C 180,E1 -7531.25,E2 -7531.25} C_VEL
LIN {X 0,Y 467.616,Z 413.239,A -85,B 0,C 180,E1 -7533.199,E2 -7533.199} C_VEL
LIN {X 0,Y 467.593,Z 413.242,A -85,B 0,C 180,E1 -7536.469,E2 -7536.469} C_VEL
LIN {X 0,Y 467.627,Z 413.235,A -85,B 0,C 180,E1 -7539.777,E2 -7539.777} C_VEL
LIN {X 0,Y 467.613,Z 413.239,A -85,B 0,C 180,E1 -7542.507,E2 -7542.507} C_VEL
LIN {X 0,Y 467.61,Z 413.238,A -85,B 0,C 180,E1 -7545.196,E2 -7545.196} C_VEL
LIN {X 0,Y 467.686,Z 413.228,A -85,B 0,C 180,E1 -7547.855,E2 -7547.855} C_VEL
LIN {X 0,Y 467.673,Z 413.23,A -85,B 0,C 180,E1 -7551.357,E2 -7551.357} C_VEL
LIN {X 0,Y 467.745,Z 413.223,A -85,B 0,C 180,E1 -7553.963,E2 -7553.963} C_VEL
LIN {X 0,Y 467.863,Z 413.205,A -85,B 0,C 180,E1 -7557.417,E2 -7557.417} C_VEL
LIN {X 0,Y 467.886,Z 413.205,A -85,B 0,C 180,E1 -7560,E2 -7560} C_VEL
LIN {X 0,Y 467.864,Z 413.208,A -85,B 0,C 180,E1 -7562.583,E2 -7562.583} C_VEL
LIN {X 0,Y 467.746,Z 413.222,A -85,B 0,C 180,E1 -7566.037,E2 -7566.037} C_VEL
LIN {X 0,Y 467.672,Z 413.231,A -85,B 0,C 180,E1 -7568.643,E2 -7568.643} C_VEL
LIN {X 0,Y 467.686,Z 413.23,A -85,B 0,C 180,E1 -7572.145,E2 -7572.145} C_VEL
LIN {X 0,Y 467.653,Z 413.234,A -85,B 0,C 180,E1 -7575.885,E2 -7575.885} C_VEL
LIN {X 0,Y 467.627,Z 413.235,A -85,B 0,C 180,E1 -7579.308,E2 -7579.308} C_VEL
LIN {X 0,Y 467.537,Z 413.25,A -85,B 0,C 180,E1 -7582.074,E2 -7582.074} C_VEL
LIN {X 0,Y 467.588,Z 413.24,A -85,B 0,C 180,E1 -7584.888,E2 -7584.888} C_VEL
LIN {X 0,Y 467.63,Z 413.238,A -85,B 0,C 180,E1 -7587.768,E2 -7587.768} C_VEL
LIN {X 0,Y 467.572,Z 413.242,A -85,B 0,C 180,E1 -7591.045,E2 -7591.045} C_VEL
LIN {X 0,Y 467.592,Z 413.242,A -85,B 0,C 180,E1 -7594.243,E2 -7594.243} C_VEL
LIN {X 0,Y 467.553,Z 413.245,A -85,B 0,C 180,E1 -7597.187,E2 -7597.187} C_VEL
LIN {X 0,Y 467.581,Z 413.243,A -85,B 0,C 180,E1 -7600.264,E2 -7600.264} C_VEL
LIN {X 0,Y 467.588,Z 413.245,A -85,B 0,C 180,E1 -7602.567,E2 -7602.567} C_VEL
LIN {X 0,Y 467.573,Z 413.246,A -85,B 0,C 180,E1 -7605.053,E2 -7605.053} C_VEL
LIN {X 0,Y 467.591,Z 413.241,A -85,B 0,C 180,E1 -7607.44,E2 -7607.44} C_VEL
LIN {X 0,Y 467.646,Z 413.293,A -85,B 0,C 180,E1 -7609.788,E2 -7609.788} C_VEL
LIN {X 0,Y 469.765,Z 424.188,A -85,B 0,C 180,E1 -7612.89,E2 -7612.89} C_VEL
LIN {X 0,Y 470.072,Z 427.761,A -85,B 0,C 180,E1 -7613.838,E2 -7613.838} C_VEL
LIN {X 0,Y 469.356,Z 442.04,A -85,B 0,C 180,E1 -7617.381,E2 -7617.381} C_VEL
LIN {X 0,Y 468.916,Z 454.589,A -85,B 0,C 180,E1 -7620.377,E2 -7620.377} C_VEL
LIN {X 0,Y 468.483,Z 468.009,A -85,B 0,C 180,E1 -7623.494,E2 -7623.494} C_VEL
LIN {X 0,Y 468.112,Z 481.924,A -85,B 0,C 180,E1 -7626.671,E2 -7626.671} C_VEL
LIN {X 0,Y 467.724,Z 496.656,A -85,B 0,C 180,E1 -7630.011,E2 -7630.011} C_VEL
LIN {X 0,Y 467.388,Z 509.601,A -85,B 0,C 180,E1 -7632.949,E2 -7632.949} C_VEL
LIN {X 0,Y 467.289,Z 516.582,A -85,B 0,C 180,E1 -7634.545,E2 -7634.545} C_VEL
LIN {X 0,Y 468.723,Z 532.206,A -85,B 0,C 180,E1 -7634.983,E2 -7634.983} C_VEL
LIN {X 0,Y 469.702,Z 541.855,A -85,B 0,C 180,E1 -7635.375,E2 -7635.375} C_VEL
LIN {X 0,Y 469.279,Z 552.988,A -85,B 0,C 180,E1 -7635.915,E2 -7635.915} C_VEL
LIN {X 0,Y 468.775,Z 564.987,A -85,B 0,C 180,E1 -7636.673,E2 -7636.673} C_VEL
LIN {X 0,Y 468.341,Z 576.028,A -85,B 0,C 180,E1 -7637.566,E2 -7637.566} C_VEL
LIN {X 0,Y 467.86,Z 585.638,A -85,B 0,C 180,E1 -7638.519,E2 -7638.519} C_VEL
LIN {X 0,Y 467.487,Z 594.658,A -85,B 0,C 180,E1 -7639.607,E2 -7639.607} C_VEL
LIN {X 0,Y 467.22,Z 603.491,A -85,B 0,C 180,E1 -7640.913,E2 -7640.913} C_VEL
LIN {X 0,Y 467.036,Z 610.565,A -85,B 0,C 180,E1 -7642.216,E2 -7642.216} C_VEL
LIN {X 0,Y 466.962,Z 616.823,A -85,B 0,C 180,E1 -7643.667,E2 -7643.667} C_VEL
LIN {X 0,Y 466.954,Z 621.988,A -85,B 0,C 180,E1 -7645.252,E2 -7645.252} C_VEL
LIN {X 0,Y 466.96,Z 625.014,A -85,B 0,C 180,E1 -7646.549,E2 -7646.549} C_VEL
LIN {X 0,Y 466.95,Z 626.454,A -85,B 0,C 180,E1 -7647.412,E2 -7647.412} C_VEL
LIN {X 0,Y 466.924,Z 627.479,A -85,B 0,C 180,E1 -7648.275,E2 -7648.275} C_VEL
LIN {X 0,Y 467.019,Z 628.344,A -85,B 0,C 180,E1 -7650,E2 -7650} C_VEL
LIN {X 0,Y 466.924,Z 627.481,A -85,B 0,C 180,E1 -7651.725,E2 -7651.725} C_VEL
LIN {X 0,Y 466.95,Z 626.458,A -85,B 0,C 180,E1 -7652.588,E2 -7652.588} C_VEL
LIN {X 0,Y 466.96,Z 625.018,A -85,B 0,C 180,E1 -7653.452,E2 -7653.452} C_VEL
LIN {X 0,Y 466.954,Z 621.989,A -85,B 0,C 180,E1 -7654.748,E2 -7654.748} C_VEL
LIN {X 0,Y 466.961,Z 616.823,A -85,B 0,C 180,E1 -7656.332,E2 -7656.332} C_VEL
LIN {X 0,Y 467.037,Z 610.565,A -85,B 0,C 180,E1 -7657.784,E2 -7657.784} C_VEL
LIN {X 0,Y 467.22,Z 603.492,A -85,B 0,C 180,E1 -7659.088,E2 -7659.088} C_VEL
LIN {X 0,Y 467.487,Z 594.658,A -85,B 0,C 180,E1 -7660.393,E2 -7660.393} C_VEL
LIN {X 0,Y 467.829,Z 585.632,A -85,B 0,C 180,E1 -7661.481,E2 -7661.481} C_VEL
LIN {X 0,Y 468.305,Z 576.344,A -85,B 0,C 180,E1 -7662.405,E2 -7662.405} C_VEL
LIN {X 0,Y 468.778,Z 564.987,A -85,B 0,C 180,E1 -7663.327,E2 -7663.327} C_VEL
LIN {X 0,Y 469.272,Z 552.977,A -85,B 0,C 180,E1 -7664.085,E2 -7664.085} C_VEL
LIN {X 0,Y 469.668,Z 540.513,A -85,B 0,C 180,E1 -7664.682,E2 -7664.682} C_VEL
LIN {X 0,Y 468.548,Z 529.383,A -85,B 0,C 180,E1 -7665.107,E2 -7665.107} C_VEL
LIN {X 0,Y 467.289,Z 516.557,A -85,B 0,C 180,E1 -7665.456,E2 -7665.456} C_VEL
LIN {X 0,Y 467.623,Z 502.057,A -85,B 0,C 180,E1 -7668.766,E2 -7668.766} C_VEL
LIN {X 0,Y 467.968,Z 486.512,A -85,B 0,C 180,E1 -7672.285,E2 -7672.285} C_VEL
LIN {X 0,Y 468.415,Z 471.107,A -85,B 0,C 180,E1 -7675.792,E2 -7675.792} C_VEL
LIN {X 0,Y 468.836,Z 456.607,A -85,B 0,C 180,E1 -7679.146,E2 -7679.146} C_VEL
LIN {X 0,Y 469.282,Z 444.091,A -85,B 0,C 180,E1 -7682.117,E2 -7682.117} C_VEL
LIN {X 0,Y 469.978,Z 429.644,A -85,B 0,C 180,E1 -7685.676,E2 -7685.676} C_VEL
LIN {X 0,Y 469.942,Z 425.531,A -85,B 0,C 180,E1 -7686.741,E2 -7686.741} C_VEL
LIN {X 0,Y 467.807,Z 414.031,A -85,B 0,C 180,E1 -7689.987,E2 -7689.987} C_VEL
LIN {X 0,Y 467.626,Z 413.236,A -85,B 0,C 180,E1 -7690.26,E2 -7690.26} C_VEL
LIN {X 0,Y 467.589,Z 413.244,A -85,B 0,C 180,E1 -7692.567,E2 -7692.567} C_VEL
LIN {X 0,Y 467.574,Z 413.244,A -85,B 0,C 180,E1 -7695.053,E2 -7695.053} C_VEL
LIN {X 0,Y 467.592,Z 413.242,A -85,B 0,C 180,E1 -7697.44,E2 -7697.44} C_VEL
LIN {X 0,Y 467.585,Z 413.241,A -85,B 0,C 180,E1 -7700.855,E2 -7700.855} C_VEL
LIN {X 0,Y 467.566,Z 413.245,A -85,B 0,C 180,E1 -7704.26,E2 -7704.26} C_VEL
LIN {X 0,Y 467.586,Z 413.241,A -85,B 0,C 180,E1 -7707.321,E2 -7707.321} C_VEL
LIN {X 0,Y 467.574,Z 413.242,A -85,B 0,C 180,E1 -7710.667,E2 -7710.667} C_VEL
LIN {X 0,Y 467.616,Z 413.236,A -85,B 0,C 180,E1 -7713.2,E2 -7713.2} C_VEL
LIN {X 0,Y 467.594,Z 413.241,A -85,B 0,C 180,E1 -7716.469,E2 -7716.469} C_VEL
LIN {X 0,Y 467.628,Z 413.238,A -85,B 0,C 180,E1 -7719.777,E2 -7719.777} C_VEL
LIN {X 0,Y 467.614,Z 413.237,A -85,B 0,C 180,E1 -7722.507,E2 -7722.507} C_VEL
LIN {X 0,Y 467.611,Z 413.238,A -85,B 0,C 180,E1 -7725.197,E2 -7725.197} C_VEL
LIN {X 0,Y 467.687,Z 413.23,A -85,B 0,C 180,E1 -7727.855,E2 -7727.855} C_VEL
LIN {X 0,Y 467.673,Z 413.231,A -85,B 0,C 180,E1 -7731.357,E2 -7731.357} C_VEL
LIN {X 0,Y 467.747,Z 413.222,A -85,B 0,C 180,E1 -7733.963,E2 -7733.963} C_VEL
LIN {X 0,Y 467.865,Z 413.208,A -85,B 0,C 180,E1 -7737.417,E2 -7737.417} C_VEL
LIN {X 0,Y 467.887,Z 413.205,A -85,B 0,C 180,E1 -7740,E2 -7740} C_VEL
LIN {X 0,Y 467.864,Z 413.205,A -85,B 0,C 180,E1 -7742.583,E2 -7742.583} C_VEL
LIN {X 0,Y 467.741,Z 413.223,A -85,B 0,C 180,E1 -7746.037,E2 -7746.037} C_VEL
LIN {X 0,Y 467.675,Z 413.23,A -85,B 0,C 180,E1 -7748.643,E2 -7748.643} C_VEL
LIN {X 0,Y 467.687,Z 413.228,A -85,B 0,C 180,E1 -7752.145,E2 -7752.145} C_VEL
LIN {X 0,Y 467.654,Z 413.234,A -85,B 0,C 180,E1 -7755.885,E2 -7755.885} C_VEL
LIN {X 0,Y 467.629,Z 413.238,A -85,B 0,C 180,E1 -7759.308,E2 -7759.308} C_VEL
LIN {X 0,Y 467.538,Z 413.247,A -85,B 0,C 180,E1 -7762.074,E2 -7762.074} C_VEL
LIN {X 0,Y 467.606,Z 413.24,A -85,B 0,C 180,E1 -7764.887,E2 -7764.887} C_VEL
LIN {X 0,Y 467.631,Z 413.236,A -85,B 0,C 180,E1 -7767.768,E2 -7767.768} C_VEL
LIN {X 0,Y 467.573,Z 413.245,A -85,B 0,C 180,E1 -7771.045,E2 -7771.045} C_VEL
LIN {X 0,Y 467.591,Z 413.24,A -85,B 0,C 180,E1 -7774.242,E2 -7774.242} C_VEL
LIN {X 0,Y 467.551,Z 413.248,A -85,B 0,C 180,E1 -7777.186,E2 -7777.186} C_VEL
LIN {X 0,Y 467.579,Z 413.241,A -85,B 0,C 180,E1 -7780.265,E2 -7780.265} C_VEL
